SPLINE
SPL {X  -159.661, Y  +678.114, Z    +0.000, E1    -9.575, E3 +131003.511}
SPL {X  -159.942, Y  +672.020, Z    +0.000, E1    -4.692, E3 +131022.137}
SPL {X  -160.000, Y  +664.971, Z    +0.000, E1    +0.516, E3 +131041.688}
SPL {X  -160.000, Y  +660.032, Z    +0.000, E1    +3.995, E3 +131053.631}
SPL {X  -160.000, Y  +652.280, Z    +0.000, E1    +8.913, E3 +131072.146}
SPL {X  -160.000, Y  +644.147, Z    +0.000, E1   +13.158, E3 +131095.696}
SPL {X  -160.000, Y  +641.594, Z    +0.000, E1   +13.488, E3 +131114.137}
SPL {X  -160.000, Y  +639.799, Z    +0.000, E1   +13.486, E3 +131130.047}
SPL {X  -160.000, Y  +637.896, Z    +0.000, E1   +13.493, E3 +131146.862}
SPL {X  -160.000, Y  +635.832, Z    +0.000, E1   +13.499, E3 +131165.121}
SPL {X  -160.000, Y  +633.839, Z    +0.000, E1   +13.489, E3 +131182.810}
SPL {X  -160.000, Y  +631.625, Z    +0.000, E1   +13.508, E3 +131202.350}
SPL {X  -160.000, Y  +629.417, Z    +0.000, E1   +13.491, E3 +131221.962}
SPL {X  -160.000, Y  +627.180, Z    +0.000, E1   +13.508, E3 +131241.716}
SPL {X  -160.000, Y  +624.970, Z    +0.000, E1   +13.490, E3 +131261.366}
SPL {X  -160.000, Y  +623.020, Z    +0.000, E1   +13.491, E3 +131278.596}
SPL {X  -160.000, Y  +620.888, Z    +0.000, E1   +13.501, E3 +131297.458}
SPL {X  -160.000, Y  +618.790, Z    +0.000, E1   +13.488, E3 +131316.080}
SPL {X  -160.000, Y  +616.631, Z    +0.000, E1   +13.504, E3 +131335.134}
SPL {X  -160.000, Y  +614.230, Z    +0.000, E1   +13.510, E3 +131356.330}
SPL {X  -160.000, Y  +612.132, Z    +0.000, E1   +13.485, E3 +131375.046}
SPL {X  -160.000, Y  +610.405, Z    +0.000, E1   +13.477, E3 +131390.420}
SPL {X  -160.000, Y  +608.437, Z    +0.000, E1   +13.502, E3 +131407.675}
SPL {X  -160.000, Y  +606.281, Z    +0.000, E1   +13.502, E3 +131426.693}
SPL {X  -160.000, Y  +604.124, Z    +0.000, E1   +13.513, E3 +131445.748}
SPL {X  -160.000, Y  +601.878, Z    +0.000, E1   +13.505, E3 +131465.645}
SPL {X  -160.000, Y  +599.648, Z    +0.000, E1   +13.506, E3 +131485.422}
SPL {X  -160.000, Y  +597.673, Z    +0.000, E1   +13.479, E3 +131503.095}
SPL {X  -160.000, Y  +595.601, Z    +0.000, E1   +13.499, E3 +131521.379}
SPL {X  -160.000, Y  +593.187, Z    +0.000, E1   +13.500, E3 +131542.759}
SPL {X  -160.000, Y  +591.079, Z    +0.000, E1   +13.483, E3 +131561.485}
SPL {X  -160.000, Y  +589.151, Z    +0.000, E1   +13.489, E3 +131578.536}
SPL {X  -160.000, Y  +586.908, Z    +0.000, E1   +13.501, E3 +131598.381}
SPL {X  -160.000, Y  +584.660, Z    +0.000, E1   +13.490, E3 +131618.323}
SPL {X  -160.000, Y  +582.409, Z    +0.000, E1   +13.499, E3 +131638.241}
SPL {X  -160.000, Y  +580.150, Z    +0.000, E1   +13.490, E3 +131658.288}
SPL {X  -160.000, Y  +577.953, Z    +0.000, E1   +13.493, E3 +131677.746}
SPL {X  -160.000, Y  +575.630, Z    +0.000, E1   +13.502, E3 +131698.230}
SPL {X  -160.000, Y  +573.418, Z    +0.000, E1   +13.502, E3 +131717.738}
SPL {X  -160.000, Y  +571.226, Z    +0.000, E1   +13.520, E3 +131736.947}
SPL {X  -160.000, Y  +569.166, Z    +0.000, E1   +13.512, E3 +131755.137}
SPL {X  -160.000, Y  +567.275, Z    +0.000, E1   +13.517, E3 +131771.804}
SPL {X  -160.000, Y  +565.259, Z    +0.000, E1   +13.523, E3 +131789.593}
SPL {X  -160.000, Y  +563.305, Z    +0.000, E1   +13.512, E3 +131806.932}
SPL {X  -160.000, Y  +561.240, Z    +0.000, E1   +13.521, E3 +131825.193}
SPL {X  -160.000, Y  +558.881, Z    +0.000, E1   +13.524, E3 +131846.036}
SPL {X  -160.000, Y  +556.697, Z    +0.000, E1   +13.510, E3 +131865.422}
SPL {X  -160.000, Y  +554.624, Z    +0.000, E1   +13.512, E3 +131883.753}
SPL {X  -160.000, Y  +552.465, Z    +0.000, E1   +13.514, E3 +131902.837}
SPL {X  -160.000, Y  +550.315, Z    +0.000, E1   +13.514, E3 +131921.830}
SPL {X  -160.000, Y  +548.056, Z    +0.000, E1   +13.519, E3 +131941.831}
SPL {X  -160.000, Y  +545.826, Z    +0.000, E1   +13.501, E3 +131961.709}
SPL {X  -160.000, Y  +543.677, Z    +0.000, E1   +13.502, E3 +131980.767}
SPL {X  -160.000, Y  +541.664, Z    +0.000, E1   +13.489, E3 +131998.652}
SPL {X  -160.000, Y  +539.659, Z    +0.000, E1   +13.494, E3 +132016.413}
SPL {X  -160.000, Y  +537.370, Z    +0.000, E1   +13.501, E3 +132036.652}
SPL {X  -160.000, Y  +535.056, Z    +0.000, E1   +13.506, E3 +132057.047}
SPL {X  -160.000, Y  +532.975, Z    +0.000, E1   +13.494, E3 +132075.534}
SPL {X  -160.000, Y  +530.925, Z    +0.000, E1   +13.499, E3 +132093.696}
SPL {X  -160.000, Y  +528.768, Z    +0.000, E1   +13.498, E3 +132112.797}
SPL {X  -160.000, Y  +526.547, Z    +0.000, E1   +13.499, E3 +132132.466}
SPL {X  -160.000, Y  +523.964, Z    +0.000, E1   +13.742, E3 +132151.970}
SPL {X  -160.000, Y  +513.971, Z    +0.000, E1   +18.644, E3 +132170.882}
SPL {X  -160.000, Y  +513.562, Z    +0.000, E1   +16.972, E3 +132190.759}
SPL {X  -160.000, Y  +513.358, Z    +0.000, E1   +15.267, E3 +132211.031}
SPL {X  -160.000, Y  +512.244, Z    +0.000, E1   +14.473, E3 +132229.487}
SPL {X  -160.000, Y  +509.675, Z    +0.000, E1   +14.481, E3 +132250.631}
SPL {X  -160.000, Y  +507.162, Z    +0.000, E1   +14.470, E3 +132271.371}
SPL {X  -160.000, Y  +504.735, Z    +0.000, E1   +14.473, E3 +132291.342}
SPL {X  -160.000, Y  +502.261, Z    +0.000, E1   +14.476, E3 +132311.678}
SPL {X  -160.000, Y  +499.798, Z    +0.000, E1   +14.482, E3 +132331.880}
SPL {X  -160.000, Y  +497.435, Z    +0.000, E1   +14.476, E3 +132351.357}
SPL {X  -160.000, Y  +495.089, Z    +0.000, E1   +14.475, E3 +132370.724}
SPL {X  -160.000, Y  +492.764, Z    +0.000, E1   +14.469, E3 +132389.895}
SPL {X  -160.000, Y  +490.292, Z    +0.000, E1   +14.476, E3 +132410.296}
SPL {X  -160.000, Y  +487.641, Z    +0.000, E1   +14.470, E3 +132432.192}
SPL {X  -160.000, Y  +485.054, Z    +0.000, E1   +14.460, E3 +132453.635}
SPL {X  -160.000, Y  +482.421, Z    +0.000, E1   +14.461, E3 +132475.353}
SPL {X  -160.000, Y  +480.000, Z    +0.000, E1   +14.451, E3 +132495.318}
SPL {X  -160.000, Y  +477.551, Z    +0.000, E1   +14.466, E3 +132515.446}
SPL {X  -160.000, Y  +475.253, Z    +0.000, E1   +14.450, E3 +132534.420}
SPL {X  -160.000, Y  +473.070, Z    +0.000, E1   +14.454, E3 +132552.441}
SPL {X  -160.000, Y  +470.603, Z    +0.000, E1   +14.464, E3 +132572.741}
SPL {X  -160.000, Y  +468.243, Z    +0.000, E1   +14.458, E3 +132592.141}
SPL {X  -160.000, Y  +465.791, Z    +0.000, E1   +14.475, E3 +132612.285}
SPL {X  -160.000, Y  +463.103, Z    +0.000, E1   +14.474, E3 +132634.433}
SPL {X  -160.000, Y  +460.743, Z    +0.000, E1   +14.465, E3 +132653.842}
SPL {X  -160.000, Y  +458.292, Z    +0.000, E1   +14.492, E3 +132673.841}
SPL {X  -160.000, Y  +455.874, Z    +0.000, E1   +14.484, E3 +132693.699}
SPL {X  -160.000, Y  +453.555, Z    +0.000, E1   +14.488, E3 +132712.778}
SPL {X  -160.000, Y  +451.093, Z    +0.000, E1   +14.485, E3 +132733.090}
SPL {X  -160.000, Y  +448.700, Z    +0.000, E1   +14.483, E3 +132752.779}
SPL {X  -160.000, Y  +446.277, Z    +0.000, E1   +14.485, E3 +132772.703}
SPL {X  -160.000, Y  +443.879, Z    +0.000, E1   +14.485, E3 +132792.441}
SPL {X  -160.000, Y  +441.447, Z    +0.000, E1   +14.485, E3 +132812.448}
SPL {X  -160.000, Y  +439.006, Z    +0.000, E1   +14.488, E3 +132832.531}
SPL {X  -160.000, Y  +436.311, Z    +0.000, E1   +14.498, E3 +132854.690}
SPL {X  -160.000, Y  +433.559, Z    +0.000, E1   +14.491, E3 +132877.360}
SPL {X  -160.000, Y  +431.162, Z    +0.000, E1   +14.479, E3 +132897.111}
SPL {X  -160.000, Y  +429.152, Z    +0.000, E1   +14.469, E3 +132913.692}
SPL {X  -160.000, Y  +426.863, Z    +0.000, E1   +14.490, E3 +132932.471}
SPL {X  -160.000, Y  +424.653, Z    +0.000, E1   +14.467, E3 +132950.731}
SPL {X  -160.000, Y  +422.337, Z    +0.000, E1   +14.492, E3 +132969.715}
SPL {X  -160.000, Y  +419.639, Z    +0.000, E1   +14.504, E3 +132991.755}
SPL {X  -160.000, Y  +417.127, Z    +0.000, E1   +14.501, E3 +133012.346}
SPL {X  -160.000, Y  +414.849, Z    +0.000, E1   +14.496, E3 +133031.080}
SPL {X  -160.000, Y  +412.396, Z    +0.000, E1   +14.505, E3 +133051.269}
SPL {X  -160.000, Y  +409.815, Z    +0.000, E1   +14.498, E3 +133072.523}
SPL {X  -160.000, Y  +407.614, Z    +0.000, E1   +14.484, E3 +133090.649}
SPL {X  -160.000, Y  +405.406, Z    +0.000, E1   +14.501, E3 +133108.712}
SPL {X  -160.000, Y  +402.958, Z    +0.000, E1   +14.500, E3 +133128.882}
SPL {X  -160.000, Y  +400.690, Z    +0.000, E1   +14.484, E3 +133147.593}
SPL {X  -160.000, Y  +398.391, Z    +0.000, E1   +14.502, E3 +133166.419}
SPL {X  -160.000, Y  +395.999, Z    +0.000, E1   +14.484, E3 +133186.209}
SPL {X  -160.000, Y  +393.685, Z    +0.000, E1   +14.486, E3 +133205.282}
SPL {X  -159.999, Y  +391.313, Z    +0.000, E1   +14.479, E3 +133224.864}
SPL {X  -159.970, Y  +388.900, Z    +0.000, E1   +14.480, E3 +133244.748}
SPL {X  -159.903, Y  +386.417, Z    +0.000, E1   +14.475, E3 +133265.253}
SPL {X  -159.796, Y  +383.921, Z    +0.000, E1   +14.466, E3 +133285.909}
SPL {X  -159.651, Y  +381.443, Z    +0.000, E1   +14.453, E3 +133306.456}
SPL {X  -159.474, Y  +379.042, Z    +0.000, E1   +14.434, E3 +133326.420}
SPL {X  -159.316, Y  +377.219, Z    +0.000, E1   +14.400, E3 +133341.649}
ENDSPLINE

SPLINE
SPL {X  -159.452, Y  +378.767, Z    +0.000, E1   +11.887, E3 +133362.638}
SPL {X  -159.840, Y  +384.856, Z    +0.000, E1    +7.126, E3 +133381.609}
SPL {X  -159.991, Y  +390.336, Z    +0.000, E1    +2.803, E3 +133395.432}
SPL {X  -160.000, Y  +403.532, Z    +0.000, E1    -6.523, E3 +133413.153}
SPL {X  -160.000, Y  +409.023, Z    +0.000, E1   -10.003, E3 +133423.926}
SPL {X  -160.000, Y  +418.032, Z    +0.000, E1   -14.569, E3 +133448.786}
SPL {X  -160.000, Y  +420.561, Z    +0.000, E1   -14.816, E3 +133466.266}
SPL {X  -160.000, Y  +422.801, Z    +0.000, E1   -14.823, E3 +133484.214}
SPL {X  -160.000, Y  +425.518, Z    +0.000, E1   -14.845, E3 +133505.989}
SPL {X  -160.000, Y  +428.688, Z    +0.000, E1   -14.854, E3 +133531.397}
SPL {X  -160.000, Y  +431.971, Z    +0.000, E1   -14.849, E3 +133557.866}
SPL {X  -160.000, Y  +435.345, Z    +0.000, E1   -14.857, E3 +133584.916}
SPL {X  -160.000, Y  +438.732, Z    +0.000, E1   -14.858, E3 +133612.064}
SPL {X  -160.000, Y  +441.925, Z    +0.000, E1   -14.848, E3 +133637.734}
SPL {X  -160.000, Y  +444.299, Z    +0.000, E1   -14.809, E3 +133656.919}
SPL {X  -160.000, Y  +446.229, Z    +0.000, E1   -14.820, E3 +133672.338}
SPL {X  -160.000, Y  +448.987, Z    +0.000, E1   -14.868, E3 +133694.275}
SPL {X  -160.000, Y  +452.351, Z    +0.000, E1   -14.871, E3 +133721.251}
SPL {X  -160.000, Y  +455.709, Z    +0.000, E1   -14.880, E3 +133748.065}
SPL {X  -160.000, Y  +458.189, Z    +0.000, E1   -14.832, E3 +133768.067}
SPL {X  -160.000, Y  +459.885, Z    +0.000, E1   -14.825, E3 +133781.737}
SPL {X  -160.000, Y  +462.438, Z    +0.000, E1   -14.868, E3 +133802.147}
SPL {X  -160.000, Y  +465.575, Z    +0.000, E1   -14.849, E3 +133827.456}
SPL {X  -160.000, Y  +468.581, Z    +0.000, E1   -14.841, E3 +133851.688}
SPL {X  -160.000, Y  +471.795, Z    +0.000, E1   -14.854, E3 +133877.475}
SPL {X  -160.000, Y  +475.138, Z    +0.000, E1   -14.853, E3 +133904.326}
SPL {X  -160.000, Y  +477.981, Z    +0.000, E1   -14.823, E3 +133927.246}
SPL {X  -160.000, Y  +480.658, Z    +0.000, E1   -14.835, E3 +133948.722}
SPL {X  -160.000, Y  +483.534, Z    +0.000, E1   -14.838, E3 +133971.817}
SPL {X  -160.000, Y  +486.226, Z    +0.000, E1   -14.823, E3 +133993.482}
SPL {X  -160.000, Y  +488.751, Z    +0.000, E1   -14.827, E3 +134013.754}
SPL {X  -160.000, Y  +491.612, Z    +0.000, E1   -14.844, E3 +134036.677}
SPL {X  -160.000, Y  +494.417, Z    +0.000, E1   -14.827, E3 +134059.268}
SPL {X  -160.000, Y  +496.961, Z    +0.000, E1   -14.824, E3 +134079.712}
SPL {X  -160.000, Y  +499.610, Z    +0.000, E1   -14.830, E3 +134100.984}
SPL {X  -160.000, Y  +502.268, Z    +0.000, E1   -14.832, E3 +134122.254}
SPL {X  -160.000, Y  +505.041, Z    +0.000, E1   -14.849, E3 +134144.416}
SPL {X  -160.000, Y  +507.743, Z    +0.000, E1   -14.842, E3 +134166.040}
SPL {X  -160.000, Y  +510.437, Z    +0.000, E1   -14.860, E3 +134187.554}
SPL {X  -160.000, Y  +513.179, Z    +0.000, E1   -14.849, E3 +134209.601}
SPL {X  -160.000, Y  +515.613, Z    +0.000, E1   -14.829, E3 +134229.272}
SPL {X  -160.000, Y  +518.188, Z    +0.000, E1   -14.845, E3 +134249.901}
SPL {X  -160.000, Y  +520.790, Z    +0.000, E1   -14.839, E3 +134270.730}
SPL {X  -160.000, Y  +523.469, Z    +0.000, E1   -14.855, E3 +134292.178}
SPL {X  -160.000, Y  +526.403, Z    +0.000, E1   -14.858, E3 +134315.714}
SPL {X  -160.000, Y  +529.266, Z    +0.000, E1   -14.848, E3 +134338.722}
SPL {X  -160.000, Y  +531.688, Z    +0.000, E1   -14.826, E3 +134358.271}
SPL {X  -160.000, Y  +534.214, Z    +0.000, E1   -14.841, E3 +134378.534}
SPL {X  -160.000, Y  +537.002, Z    +0.000, E1   -14.839, E3 +134400.953}
SPL {X  -160.000, Y  +539.729, Z    +0.000, E1   -14.840, E3 +134422.764}
SPL {X  -160.000, Y  +542.408, Z    +0.000, E1   -14.839, E3 +134444.317}
SPL {X  -160.000, Y  +545.014, Z    +0.000, E1   -14.831, E3 +134465.262}
SPL {X  -160.000, Y  +547.659, Z    +0.000, E1   -14.839, E3 +134486.477}
SPL {X  -160.000, Y  +550.215, Z    +0.000, E1   -14.827, E3 +134507.042}
SPL {X  -160.000, Y  +552.762, Z    +0.000, E1   -14.836, E3 +134527.460}
SPL {X  -160.000, Y  +555.331, Z    +0.000, E1   -14.837, E3 +134548.001}
SPL {X  -160.000, Y  +558.235, Z    +0.000, E1   -14.869, E3 +134571.165}
SPL {X  -160.000, Y  +561.088, Z    +0.000, E1   -14.848, E3 +134594.083}
SPL {X  -160.000, Y  +563.693, Z    +0.000, E1   -14.852, E3 +134614.944}
SPL {X  -160.000, Y  +566.560, Z    +0.000, E1   -14.865, E3 +134637.921}
SPL {X  -160.000, Y  +569.305, Z    +0.000, E1   -14.848, E3 +134659.950}
SPL {X  -160.000, Y  +571.769, Z    +0.000, E1   -14.852, E3 +134679.696}
SPL {X  -160.000, Y  +574.366, Z    +0.000, E1   -14.855, E3 +134700.483}
SPL {X  -160.000, Y  +577.037, Z    +0.000, E1   -14.859, E3 +134721.882}
SPL {X  -160.000, Y  +579.855, Z    +0.000, E1   -14.869, E3 +134744.409}
SPL {X  -160.000, Y  +582.456, Z    +0.000, E1   -14.854, E3 +134765.269}
SPL {X  -160.000, Y  +585.083, Z    +0.000, E1   -14.866, E3 +134786.319}
SPL {X  -160.000, Y  +587.675, Z    +0.000, E1   -14.853, E3 +134807.110}
SPL {X  -160.000, Y  +590.216, Z    +0.000, E1   -14.864, E3 +134827.429}
SPL {X  -160.000, Y  +592.848, Z    +0.000, E1   -14.865, E3 +134848.480}
SPL {X  -160.000, Y  +595.342, Z    +0.000, E1   -14.848, E3 +134868.658}
SPL {X  -160.000, Y  +597.995, Z    +0.000, E1   -14.848, E3 +134889.998}
SPL {X  -160.000, Y  +600.731, Z    +0.000, E1   -14.846, E3 +134911.949}
SPL {X  -160.000, Y  +603.404, Z    +0.000, E1   -14.846, E3 +134933.385}
SPL {X  -160.000, Y  +605.923, Z    +0.000, E1   -14.838, E3 +134953.626}
SPL {X  -160.000, Y  +608.492, Z    +0.000, E1   -14.846, E3 +134974.230}
SPL {X  -160.000, Y  +611.345, Z    +0.000, E1   -14.856, E3 +134997.088}
SPL {X  -160.000, Y  +614.087, Z    +0.000, E1   -14.839, E3 +135019.147}
SPL {X  -160.000, Y  +616.566, Z    +0.000, E1   -14.839, E3 +135039.041}
SPL {X  -160.000, Y  +619.350, Z    +0.000, E1   -14.855, E3 +135061.329}
SPL {X  -160.000, Y  +622.198, Z    +0.000, E1   -14.846, E3 +135084.213}
SPL {X  -160.000, Y  +624.642, Z    +0.000, E1   -14.829, E3 +135103.886}
SPL {X  -160.000, Y  +627.119, Z    +0.000, E1   -14.843, E3 +135123.726}
SPL {X  -160.000, Y  +629.682, Z    +0.000, E1   -14.838, E3 +135144.295}
SPL {X  -160.000, Y  +632.223, Z    +0.000, E1   -14.841, E3 +135164.686}
SPL {X  -160.000, Y  +634.941, Z    +0.000, E1   -14.846, E3 +135186.484}
SPL {X  -160.000, Y  +637.723, Z    +0.000, E1   -14.844, E3 +135208.828}
SPL {X  -160.000, Y  +640.315, Z    +0.000, E1   -14.836, E3 +135229.626}
SPL {X  -160.000, Y  +643.085, Z    +0.000, E1   -14.865, E3 +135251.677}
SPL {X  -160.000, Y  +645.845, Z    +0.000, E1   -14.848, E3 +135273.865}
SPL {X  -160.000, Y  +648.229, Z    +0.000, E1   -14.834, E3 +135293.075}
SPL {X  -160.000, Y  +650.656, Z    +0.000, E1   -14.835, E3 +135312.631}
SPL {X  -160.000, Y  +653.134, Z    +0.000, E1   -14.827, E3 +135332.558}
SPL {X  -160.000, Y  +655.670, Z    +0.000, E1   -14.841, E3 +135352.852}
SPL {X  -160.000, Y  +658.349, Z    +0.000, E1   -14.842, E3 +135374.328}
SPL {X  -160.000, Y  +660.936, Z    +0.000, E1   -14.838, E3 +135395.080}
SPL {X  -160.000, Y  +663.567, Z    +0.000, E1   -14.845, E3 +135416.210}
SPL {X  -160.000, Y  +666.216, Z    +0.000, E1   -14.832, E3 +135437.527}
SPL {X  -159.997, Y  +668.731, Z    +0.000, E1   -14.834, E3 +135457.719}
SPL {X  -159.962, Y  +671.176, Z    +0.000, E1   -14.822, E3 +135477.430}
SPL {X  -159.895, Y  +673.507, Z    +0.000, E1   -14.821, E3 +135496.161}
SPL {X  -159.785, Y  +675.985, Z    +0.000, E1   -14.818, E3 +135516.163}
SPL {X  -159.627, Y  +678.622, Z    +0.000, E1   -14.804, E3 +135537.516}
SPL {X  -159.438, Y  +681.094, Z    +0.000, E1   -14.770, E3 +135557.687}
SPL {X  -159.262, Y  +683.054, Z    +0.000, E1   -14.719, E3 +135573.915}
ENDSPLINE

SPLINE
SPL {X  -159.661, Y  +678.114, Z    +0.000, E1    -9.575, E3 +135603.507}
SPL {X  -159.942, Y  +672.020, Z    +0.000, E1    -4.692, E3 +135622.134}
SPL {X  -160.000, Y  +664.971, Z    +0.000, E1    +0.516, E3 +135641.684}
SPL {X  -160.000, Y  +660.032, Z    +0.000, E1    +3.995, E3 +135653.627}
SPL {X  -160.000, Y  +652.280, Z    +0.000, E1    +8.913, E3 +135672.142}
SPL {X  -160.000, Y  +644.147, Z    +0.000, E1   +13.158, E3 +135695.693}
SPL {X  -160.000, Y  +641.594, Z    +0.000, E1   +13.488, E3 +135714.134}
SPL {X  -160.000, Y  +639.799, Z    +0.000, E1   +13.486, E3 +135730.044}
SPL {X  -160.000, Y  +637.896, Z    +0.000, E1   +13.493, E3 +135746.859}
SPL {X  -160.000, Y  +635.832, Z    +0.000, E1   +13.499, E3 +135765.118}
SPL {X  -160.000, Y  +633.839, Z    +0.000, E1   +13.489, E3 +135782.806}
SPL {X  -160.000, Y  +631.625, Z    +0.000, E1   +13.508, E3 +135802.347}
SPL {X  -160.000, Y  +629.417, Z    +0.000, E1   +13.491, E3 +135821.959}
SPL {X  -160.000, Y  +627.180, Z    +0.000, E1   +13.508, E3 +135841.713}
SPL {X  -160.000, Y  +624.970, Z    +0.000, E1   +13.490, E3 +135861.363}
SPL {X  -160.000, Y  +623.020, Z    +0.000, E1   +13.491, E3 +135878.592}
SPL {X  -160.000, Y  +620.888, Z    +0.000, E1   +13.501, E3 +135897.455}
SPL {X  -160.000, Y  +618.790, Z    +0.000, E1   +13.488, E3 +135916.077}
SPL {X  -160.000, Y  +616.631, Z    +0.000, E1   +13.504, E3 +135935.131}
SPL {X  -160.000, Y  +614.230, Z    +0.000, E1   +13.510, E3 +135956.327}
SPL {X  -160.000, Y  +612.132, Z    +0.000, E1   +13.485, E3 +135975.043}
SPL {X  -160.000, Y  +610.405, Z    +0.000, E1   +13.477, E3 +135990.416}
SPL {X  -160.000, Y  +608.437, Z    +0.000, E1   +13.502, E3 +136007.672}
SPL {X  -160.000, Y  +606.281, Z    +0.000, E1   +13.502, E3 +136026.689}
SPL {X  -160.000, Y  +604.124, Z    +0.000, E1   +13.513, E3 +136045.745}
SPL {X  -160.000, Y  +601.878, Z    +0.000, E1   +13.505, E3 +136065.642}
SPL {X  -160.000, Y  +599.648, Z    +0.000, E1   +13.506, E3 +136085.419}
SPL {X  -160.000, Y  +597.673, Z    +0.000, E1   +13.479, E3 +136103.092}
SPL {X  -160.000, Y  +595.601, Z    +0.000, E1   +13.499, E3 +136121.375}
SPL {X  -160.000, Y  +593.187, Z    +0.000, E1   +13.500, E3 +136142.755}
SPL {X  -160.000, Y  +591.079, Z    +0.000, E1   +13.483, E3 +136161.482}
SPL {X  -160.000, Y  +589.151, Z    +0.000, E1   +13.489, E3 +136178.533}
SPL {X  -160.000, Y  +586.908, Z    +0.000, E1   +13.501, E3 +136198.378}
SPL {X  -160.000, Y  +584.660, Z    +0.000, E1   +13.490, E3 +136218.320}
SPL {X  -160.000, Y  +582.409, Z    +0.000, E1   +13.499, E3 +136238.238}
SPL {X  -160.000, Y  +580.150, Z    +0.000, E1   +13.490, E3 +136258.284}
SPL {X  -160.000, Y  +577.953, Z    +0.000, E1   +13.493, E3 +136277.743}
SPL {X  -160.000, Y  +575.630, Z    +0.000, E1   +13.502, E3 +136298.227}
SPL {X  -160.000, Y  +573.418, Z    +0.000, E1   +13.502, E3 +136317.735}
SPL {X  -160.000, Y  +571.226, Z    +0.000, E1   +13.520, E3 +136336.943}
SPL {X  -160.000, Y  +569.166, Z    +0.000, E1   +13.512, E3 +136355.134}
SPL {X  -160.000, Y  +567.275, Z    +0.000, E1   +13.517, E3 +136371.801}
SPL {X  -160.000, Y  +565.259, Z    +0.000, E1   +13.523, E3 +136389.590}
SPL {X  -160.000, Y  +563.305, Z    +0.000, E1   +13.512, E3 +136406.929}
SPL {X  -160.000, Y  +561.240, Z    +0.000, E1   +13.521, E3 +136425.190}
SPL {X  -160.000, Y  +558.881, Z    +0.000, E1   +13.524, E3 +136446.032}
SPL {X  -160.000, Y  +556.697, Z    +0.000, E1   +13.510, E3 +136465.418}
SPL {X  -160.000, Y  +554.624, Z    +0.000, E1   +13.512, E3 +136483.749}
SPL {X  -160.000, Y  +552.465, Z    +0.000, E1   +13.514, E3 +136502.834}
SPL {X  -160.000, Y  +550.315, Z    +0.000, E1   +13.514, E3 +136521.827}
SPL {X  -160.000, Y  +548.056, Z    +0.000, E1   +13.519, E3 +136541.828}
SPL {X  -160.000, Y  +545.826, Z    +0.000, E1   +13.501, E3 +136561.706}
SPL {X  -160.000, Y  +543.677, Z    +0.000, E1   +13.502, E3 +136580.764}
SPL {X  -160.000, Y  +541.664, Z    +0.000, E1   +13.489, E3 +136598.649}
SPL {X  -160.000, Y  +539.659, Z    +0.000, E1   +13.494, E3 +136616.409}
SPL {X  -160.000, Y  +537.370, Z    +0.000, E1   +13.501, E3 +136636.648}
SPL {X  -160.000, Y  +535.056, Z    +0.000, E1   +13.506, E3 +136657.044}
SPL {X  -160.000, Y  +532.975, Z    +0.000, E1   +13.494, E3 +136675.531}
SPL {X  -160.000, Y  +530.925, Z    +0.000, E1   +13.499, E3 +136693.692}
SPL {X  -160.000, Y  +528.768, Z    +0.000, E1   +13.498, E3 +136712.794}
SPL {X  -160.000, Y  +526.547, Z    +0.000, E1   +13.499, E3 +136732.462}
SPL {X  -160.000, Y  +523.964, Z    +0.000, E1   +13.742, E3 +136751.967}
SPL {X  -160.000, Y  +513.971, Z    +0.000, E1   +18.644, E3 +136770.879}
SPL {X  -160.000, Y  +513.562, Z    +0.000, E1   +16.972, E3 +136790.756}
SPL {X  -160.000, Y  +513.358, Z    +0.000, E1   +15.267, E3 +136811.028}
SPL {X  -160.000, Y  +512.244, Z    +0.000, E1   +14.473, E3 +136829.484}
SPL {X  -160.000, Y  +509.675, Z    +0.000, E1   +14.481, E3 +136850.627}
SPL {X  -160.000, Y  +507.162, Z    +0.000, E1   +14.470, E3 +136871.367}
SPL {X  -160.000, Y  +504.735, Z    +0.000, E1   +14.473, E3 +136891.339}
SPL {X  -160.000, Y  +502.261, Z    +0.000, E1   +14.476, E3 +136911.675}
SPL {X  -160.000, Y  +499.798, Z    +0.000, E1   +14.482, E3 +136931.877}
SPL {X  -160.000, Y  +497.435, Z    +0.000, E1   +14.476, E3 +136951.354}
SPL {X  -160.000, Y  +495.089, Z    +0.000, E1   +14.475, E3 +136970.721}
SPL {X  -160.000, Y  +492.764, Z    +0.000, E1   +14.469, E3 +136989.892}
SPL {X  -160.000, Y  +490.292, Z    +0.000, E1   +14.476, E3 +137010.293}
SPL {X  -160.000, Y  +487.641, Z    +0.000, E1   +14.470, E3 +137032.189}
SPL {X  -160.000, Y  +485.054, Z    +0.000, E1   +14.460, E3 +137053.632}
SPL {X  -160.000, Y  +482.421, Z    +0.000, E1   +14.461, E3 +137075.350}
SPL {X  -160.000, Y  +480.000, Z    +0.000, E1   +14.451, E3 +137095.314}
SPL {X  -160.000, Y  +477.551, Z    +0.000, E1   +14.466, E3 +137115.443}
SPL {X  -160.000, Y  +475.253, Z    +0.000, E1   +14.450, E3 +137134.417}
SPL {X  -160.000, Y  +473.070, Z    +0.000, E1   +14.454, E3 +137152.438}
SPL {X  -160.000, Y  +470.603, Z    +0.000, E1   +14.464, E3 +137172.738}
SPL {X  -160.000, Y  +468.243, Z    +0.000, E1   +14.458, E3 +137192.137}
SPL {X  -160.000, Y  +465.791, Z    +0.000, E1   +14.475, E3 +137212.281}
SPL {X  -160.000, Y  +463.103, Z    +0.000, E1   +14.474, E3 +137234.430}
SPL {X  -160.000, Y  +460.743, Z    +0.000, E1   +14.465, E3 +137253.838}
SPL {X  -160.000, Y  +458.292, Z    +0.000, E1   +14.492, E3 +137273.838}
SPL {X  -160.000, Y  +455.874, Z    +0.000, E1   +14.484, E3 +137293.695}
SPL {X  -160.000, Y  +453.555, Z    +0.000, E1   +14.488, E3 +137312.775}
SPL {X  -160.000, Y  +451.093, Z    +0.000, E1   +14.485, E3 +137333.087}
SPL {X  -160.000, Y  +448.700, Z    +0.000, E1   +14.483, E3 +137352.776}
SPL {X  -160.000, Y  +446.277, Z    +0.000, E1   +14.485, E3 +137372.700}
SPL {X  -160.000, Y  +443.879, Z    +0.000, E1   +14.485, E3 +137392.438}
SPL {X  -160.000, Y  +441.447, Z    +0.000, E1   +14.485, E3 +137412.445}
SPL {X  -160.000, Y  +439.006, Z    +0.000, E1   +14.488, E3 +137432.528}
SPL {X  -160.000, Y  +436.311, Z    +0.000, E1   +14.498, E3 +137454.687}
SPL {X  -160.000, Y  +433.559, Z    +0.000, E1   +14.491, E3 +137477.357}
SPL {X  -160.000, Y  +431.162, Z    +0.000, E1   +14.479, E3 +137497.108}
SPL {X  -160.000, Y  +429.152, Z    +0.000, E1   +14.469, E3 +137513.689}
SPL {X  -160.000, Y  +426.863, Z    +0.000, E1   +14.490, E3 +137532.468}
SPL {X  -160.000, Y  +424.653, Z    +0.000, E1   +14.467, E3 +137550.728}
SPL {X  -160.000, Y  +422.337, Z    +0.000, E1   +14.492, E3 +137569.712}
SPL {X  -160.000, Y  +419.639, Z    +0.000, E1   +14.504, E3 +137591.752}
SPL {X  -160.000, Y  +417.127, Z    +0.000, E1   +14.501, E3 +137612.343}
SPL {X  -160.000, Y  +414.849, Z    +0.000, E1   +14.496, E3 +137631.077}
SPL {X  -160.000, Y  +412.396, Z    +0.000, E1   +14.505, E3 +137651.266}
SPL {X  -160.000, Y  +409.815, Z    +0.000, E1   +14.498, E3 +137672.520}
SPL {X  -160.000, Y  +407.614, Z    +0.000, E1   +14.484, E3 +137690.645}
SPL {X  -160.000, Y  +405.406, Z    +0.000, E1   +14.501, E3 +137708.708}
SPL {X  -160.000, Y  +402.958, Z    +0.000, E1   +14.500, E3 +137728.879}
SPL {X  -160.000, Y  +400.690, Z    +0.000, E1   +14.484, E3 +137747.590}
SPL {X  -160.000, Y  +398.391, Z    +0.000, E1   +14.502, E3 +137766.416}
SPL {X  -160.000, Y  +395.999, Z    +0.000, E1   +14.484, E3 +137786.206}
SPL {X  -160.000, Y  +393.685, Z    +0.000, E1   +14.486, E3 +137805.278}
SPL {X  -159.999, Y  +391.313, Z    +0.000, E1   +14.479, E3 +137824.860}
SPL {X  -159.970, Y  +388.900, Z    +0.000, E1   +14.480, E3 +137844.745}
SPL {X  -159.903, Y  +386.417, Z    +0.000, E1   +14.475, E3 +137865.250}
SPL {X  -159.796, Y  +383.921, Z    +0.000, E1   +14.466, E3 +137885.905}
SPL {X  -159.651, Y  +381.443, Z    +0.000, E1   +14.453, E3 +137906.453}
SPL {X  -159.474, Y  +379.042, Z    +0.000, E1   +14.434, E3 +137926.417}
SPL {X  -159.316, Y  +377.219, Z    +0.000, E1   +14.400, E3 +137941.645}
ENDSPLINE

SPLINE
SPL {X  -159.452, Y  +378.767, Z    +0.000, E1   +11.887, E3 +137962.635}
SPL {X  -159.840, Y  +384.856, Z    +0.000, E1    +7.126, E3 +137981.606}
SPL {X  -159.991, Y  +390.336, Z    +0.000, E1    +2.803, E3 +137995.429}
SPL {X  -160.000, Y  +403.532, Z    +0.000, E1    -6.523, E3 +138013.150}
SPL {X  -160.000, Y  +409.023, Z    +0.000, E1   -10.003, E3 +138023.923}
SPL {X  -160.000, Y  +418.032, Z    +0.000, E1   -14.569, E3 +138048.782}
SPL {X  -160.000, Y  +420.561, Z    +0.000, E1   -14.816, E3 +138066.263}
SPL {X  -160.000, Y  +422.801, Z    +0.000, E1   -14.823, E3 +138084.211}
SPL {X  -160.000, Y  +425.518, Z    +0.000, E1   -14.845, E3 +138105.986}
SPL {X  -160.000, Y  +428.688, Z    +0.000, E1   -14.854, E3 +138131.394}
SPL {X  -160.000, Y  +431.971, Z    +0.000, E1   -14.849, E3 +138157.862}
SPL {X  -160.000, Y  +435.345, Z    +0.000, E1   -14.857, E3 +138184.913}
SPL {X  -160.000, Y  +438.732, Z    +0.000, E1   -14.858, E3 +138212.061}
SPL {X  -160.000, Y  +441.925, Z    +0.000, E1   -14.848, E3 +138237.731}
SPL {X  -160.000, Y  +444.299, Z    +0.000, E1   -14.809, E3 +138256.916}
SPL {X  -160.000, Y  +446.229, Z    +0.000, E1   -14.820, E3 +138272.335}
SPL {X  -160.000, Y  +448.987, Z    +0.000, E1   -14.868, E3 +138294.272}
SPL {X  -160.000, Y  +452.351, Z    +0.000, E1   -14.871, E3 +138321.248}
SPL {X  -160.000, Y  +455.709, Z    +0.000, E1   -14.880, E3 +138348.062}
SPL {X  -160.000, Y  +458.189, Z    +0.000, E1   -14.832, E3 +138368.063}
SPL {X  -160.000, Y  +459.885, Z    +0.000, E1   -14.825, E3 +138381.734}
SPL {X  -160.000, Y  +462.438, Z    +0.000, E1   -14.868, E3 +138402.144}
SPL {X  -160.000, Y  +465.575, Z    +0.000, E1   -14.849, E3 +138427.452}
SPL {X  -160.000, Y  +468.581, Z    +0.000, E1   -14.841, E3 +138451.685}
SPL {X  -160.000, Y  +471.795, Z    +0.000, E1   -14.854, E3 +138477.472}
SPL {X  -160.000, Y  +475.138, Z    +0.000, E1   -14.853, E3 +138504.322}
SPL {X  -160.000, Y  +477.981, Z    +0.000, E1   -14.823, E3 +138527.243}
SPL {X  -160.000, Y  +480.658, Z    +0.000, E1   -14.835, E3 +138548.719}
SPL {X  -160.000, Y  +483.534, Z    +0.000, E1   -14.838, E3 +138571.814}
SPL {X  -160.000, Y  +486.226, Z    +0.000, E1   -14.823, E3 +138593.479}
SPL {X  -160.000, Y  +488.751, Z    +0.000, E1   -14.827, E3 +138613.751}
SPL {X  -160.000, Y  +491.612, Z    +0.000, E1   -14.844, E3 +138636.674}
SPL {X  -160.000, Y  +494.417, Z    +0.000, E1   -14.827, E3 +138659.265}
SPL {X  -160.000, Y  +496.961, Z    +0.000, E1   -14.824, E3 +138679.709}
SPL {X  -160.000, Y  +499.610, Z    +0.000, E1   -14.830, E3 +138700.981}
SPL {X  -160.000, Y  +502.268, Z    +0.000, E1   -14.832, E3 +138722.250}
SPL {X  -160.000, Y  +505.041, Z    +0.000, E1   -14.849, E3 +138744.413}
SPL {X  -160.000, Y  +507.743, Z    +0.000, E1   -14.842, E3 +138766.037}
SPL {X  -160.000, Y  +510.437, Z    +0.000, E1   -14.860, E3 +138787.551}
SPL {X  -160.000, Y  +513.179, Z    +0.000, E1   -14.849, E3 +138809.598}
SPL {X  -160.000, Y  +515.613, Z    +0.000, E1   -14.829, E3 +138829.268}
SPL {X  -160.000, Y  +518.188, Z    +0.000, E1   -14.845, E3 +138849.898}
SPL {X  -160.000, Y  +520.790, Z    +0.000, E1   -14.839, E3 +138870.727}
SPL {X  -160.000, Y  +523.469, Z    +0.000, E1   -14.855, E3 +138892.175}
SPL {X  -160.000, Y  +526.403, Z    +0.000, E1   -14.858, E3 +138915.711}
SPL {X  -160.000, Y  +529.266, Z    +0.000, E1   -14.848, E3 +138938.718}
SPL {X  -160.000, Y  +531.688, Z    +0.000, E1   -14.826, E3 +138958.268}
SPL {X  -160.000, Y  +534.214, Z    +0.000, E1   -14.841, E3 +138978.531}
SPL {X  -160.000, Y  +537.002, Z    +0.000, E1   -14.839, E3 +139000.949}
SPL {X  -160.000, Y  +539.729, Z    +0.000, E1   -14.840, E3 +139022.761}
SPL {X  -160.000, Y  +542.408, Z    +0.000, E1   -14.839, E3 +139044.314}
SPL {X  -160.000, Y  +545.014, Z    +0.000, E1   -14.831, E3 +139065.259}
SPL {X  -160.000, Y  +547.659, Z    +0.000, E1   -14.839, E3 +139086.474}
SPL {X  -160.000, Y  +550.215, Z    +0.000, E1   -14.827, E3 +139107.039}
SPL {X  -160.000, Y  +552.762, Z    +0.000, E1   -14.836, E3 +139127.457}
SPL {X  -160.000, Y  +555.331, Z    +0.000, E1   -14.837, E3 +139147.998}
SPL {X  -160.000, Y  +558.235, Z    +0.000, E1   -14.869, E3 +139171.161}
SPL {X  -160.000, Y  +561.088, Z    +0.000, E1   -14.848, E3 +139194.080}
SPL {X  -160.000, Y  +563.693, Z    +0.000, E1   -14.852, E3 +139214.940}
SPL {X  -160.000, Y  +566.560, Z    +0.000, E1   -14.865, E3 +139237.918}
SPL {X  -160.000, Y  +569.305, Z    +0.000, E1   -14.848, E3 +139259.947}
SPL {X  -160.000, Y  +571.769, Z    +0.000, E1   -14.852, E3 +139279.692}
SPL {X  -160.000, Y  +574.366, Z    +0.000, E1   -14.855, E3 +139300.479}
SPL {X  -160.000, Y  +577.037, Z    +0.000, E1   -14.859, E3 +139321.879}
SPL {X  -160.000, Y  +579.855, Z    +0.000, E1   -14.869, E3 +139344.406}
SPL {X  -160.000, Y  +582.456, Z    +0.000, E1   -14.854, E3 +139365.266}
SPL {X  -160.000, Y  +585.083, Z    +0.000, E1   -14.866, E3 +139386.316}
SPL {X  -160.000, Y  +587.675, Z    +0.000, E1   -14.853, E3 +139407.107}
SPL {X  -160.000, Y  +590.216, Z    +0.000, E1   -14.864, E3 +139427.426}
SPL {X  -160.000, Y  +592.848, Z    +0.000, E1   -14.865, E3 +139448.477}
SPL {X  -160.000, Y  +595.342, Z    +0.000, E1   -14.848, E3 +139468.655}
SPL {X  -160.000, Y  +597.995, Z    +0.000, E1   -14.848, E3 +139489.995}
SPL {X  -160.000, Y  +600.731, Z    +0.000, E1   -14.846, E3 +139511.946}
SPL {X  -160.000, Y  +603.404, Z    +0.000, E1   -14.846, E3 +139533.382}
SPL {X  -160.000, Y  +605.923, Z    +0.000, E1   -14.838, E3 +139553.623}
SPL {X  -160.000, Y  +608.492, Z    +0.000, E1   -14.846, E3 +139574.226}
SPL {X  -160.000, Y  +611.345, Z    +0.000, E1   -14.856, E3 +139597.085}
SPL {X  -160.000, Y  +614.087, Z    +0.000, E1   -14.839, E3 +139619.144}
SPL {X  -160.000, Y  +616.566, Z    +0.000, E1   -14.839, E3 +139639.038}
SPL {X  -160.000, Y  +619.350, Z    +0.000, E1   -14.855, E3 +139661.326}
SPL {X  -160.000, Y  +622.198, Z    +0.000, E1   -14.846, E3 +139684.210}
SPL {X  -160.000, Y  +624.642, Z    +0.000, E1   -14.829, E3 +139703.883}
SPL {X  -160.000, Y  +627.119, Z    +0.000, E1   -14.843, E3 +139723.723}
SPL {X  -160.000, Y  +629.682, Z    +0.000, E1   -14.838, E3 +139744.292}
SPL {X  -160.000, Y  +632.223, Z    +0.000, E1   -14.841, E3 +139764.683}
SPL {X  -160.000, Y  +634.941, Z    +0.000, E1   -14.846, E3 +139786.481}
SPL {X  -160.000, Y  +637.723, Z    +0.000, E1   -14.844, E3 +139808.825}
SPL {X  -160.000, Y  +640.315, Z    +0.000, E1   -14.836, E3 +139829.622}
SPL {X  -160.000, Y  +643.085, Z    +0.000, E1   -14.865, E3 +139851.674}
SPL {X  -160.000, Y  +645.845, Z    +0.000, E1   -14.848, E3 +139873.862}
SPL {X  -160.000, Y  +648.229, Z    +0.000, E1   -14.834, E3 +139893.072}
SPL {X  -160.000, Y  +650.656, Z    +0.000, E1   -14.835, E3 +139912.628}
SPL {X  -160.000, Y  +653.134, Z    +0.000, E1   -14.827, E3 +139932.555}
SPL {X  -160.000, Y  +655.670, Z    +0.000, E1   -14.841, E3 +139952.849}
SPL {X  -160.000, Y  +658.349, Z    +0.000, E1   -14.842, E3 +139974.325}
SPL {X  -160.000, Y  +660.936, Z    +0.000, E1   -14.838, E3 +139995.077}
SPL {X  -160.000, Y  +663.567, Z    +0.000, E1   -14.845, E3 +140016.207}
SPL {X  -160.000, Y  +666.216, Z    +0.000, E1   -14.832, E3 +140037.524}
SPL {X  -159.997, Y  +668.731, Z    +0.000, E1   -14.834, E3 +140057.716}
SPL {X  -159.962, Y  +671.176, Z    +0.000, E1   -14.822, E3 +140077.427}
SPL {X  -159.895, Y  +673.507, Z    +0.000, E1   -14.821, E3 +140096.158}
SPL {X  -159.785, Y  +675.985, Z    +0.000, E1   -14.818, E3 +140116.160}
SPL {X  -159.627, Y  +678.622, Z    +0.000, E1   -14.804, E3 +140137.512}
SPL {X  -159.438, Y  +681.094, Z    +0.000, E1   -14.770, E3 +140157.684}
SPL {X  -159.262, Y  +683.054, Z    +0.000, E1   -14.719, E3 +140173.912}
ENDSPLINE

SPLINE
SPL {X  -159.661, Y  +678.114, Z    +0.000, E1    -9.575, E3 +140203.504}
SPL {X  -159.942, Y  +672.020, Z    +0.000, E1    -4.692, E3 +140222.131}
SPL {X  -160.000, Y  +664.971, Z    +0.000, E1    +0.516, E3 +140241.681}
SPL {X  -160.000, Y  +660.032, Z    +0.000, E1    +3.995, E3 +140253.624}
SPL {X  -160.000, Y  +652.280, Z    +0.000, E1    +8.913, E3 +140272.139}
SPL {X  -160.000, Y  +644.147, Z    +0.000, E1   +13.158, E3 +140295.690}
SPL {X  -160.000, Y  +641.594, Z    +0.000, E1   +13.488, E3 +140314.131}
SPL {X  -160.000, Y  +639.799, Z    +0.000, E1   +13.486, E3 +140330.041}
SPL {X  -160.000, Y  +637.896, Z    +0.000, E1   +13.493, E3 +140346.856}
SPL {X  -160.000, Y  +635.832, Z    +0.000, E1   +13.499, E3 +140365.114}
SPL {X  -160.000, Y  +633.839, Z    +0.000, E1   +13.489, E3 +140382.803}
SPL {X  -160.000, Y  +631.625, Z    +0.000, E1   +13.508, E3 +140402.344}
SPL {X  -160.000, Y  +629.417, Z    +0.000, E1   +13.491, E3 +140421.955}
SPL {X  -160.000, Y  +627.180, Z    +0.000, E1   +13.508, E3 +140441.709}
SPL {X  -160.000, Y  +624.970, Z    +0.000, E1   +13.490, E3 +140461.359}
SPL {X  -160.000, Y  +623.020, Z    +0.000, E1   +13.491, E3 +140478.589}
SPL {X  -160.000, Y  +620.888, Z    +0.000, E1   +13.501, E3 +140497.452}
SPL {X  -160.000, Y  +618.790, Z    +0.000, E1   +13.488, E3 +140516.074}
SPL {X  -160.000, Y  +616.631, Z    +0.000, E1   +13.504, E3 +140535.128}
SPL {X  -160.000, Y  +614.230, Z    +0.000, E1   +13.510, E3 +140556.323}
SPL {X  -160.000, Y  +612.132, Z    +0.000, E1   +13.485, E3 +140575.040}
SPL {X  -160.000, Y  +610.405, Z    +0.000, E1   +13.477, E3 +140590.413}
SPL {X  -160.000, Y  +608.437, Z    +0.000, E1   +13.502, E3 +140607.669}
SPL {X  -160.000, Y  +606.281, Z    +0.000, E1   +13.502, E3 +140626.686}
SPL {X  -160.000, Y  +604.124, Z    +0.000, E1   +13.513, E3 +140645.741}
SPL {X  -160.000, Y  +601.878, Z    +0.000, E1   +13.505, E3 +140665.639}
SPL {X  -160.000, Y  +599.648, Z    +0.000, E1   +13.506, E3 +140685.415}
SPL {X  -160.000, Y  +597.673, Z    +0.000, E1   +13.479, E3 +140703.089}
SPL {X  -160.000, Y  +595.601, Z    +0.000, E1   +13.499, E3 +140721.372}
SPL {X  -160.000, Y  +593.187, Z    +0.000, E1   +13.500, E3 +140742.752}
SPL {X  -160.000, Y  +591.079, Z    +0.000, E1   +13.483, E3 +140761.478}
SPL {X  -160.000, Y  +589.151, Z    +0.000, E1   +13.489, E3 +140778.529}
SPL {X  -160.000, Y  +586.908, Z    +0.000, E1   +13.501, E3 +140798.375}
SPL {X  -160.000, Y  +584.660, Z    +0.000, E1   +13.490, E3 +140818.316}
SPL {X  -160.000, Y  +582.409, Z    +0.000, E1   +13.499, E3 +140838.235}
SPL {X  -160.000, Y  +580.150, Z    +0.000, E1   +13.490, E3 +140858.281}
SPL {X  -160.000, Y  +577.953, Z    +0.000, E1   +13.493, E3 +140877.739}
SPL {X  -160.000, Y  +575.630, Z    +0.000, E1   +13.502, E3 +140898.223}
SPL {X  -160.000, Y  +573.418, Z    +0.000, E1   +13.502, E3 +140917.731}
SPL {X  -160.000, Y  +571.226, Z    +0.000, E1   +13.520, E3 +140936.940}
SPL {X  -160.000, Y  +569.166, Z    +0.000, E1   +13.512, E3 +140955.131}
SPL {X  -160.000, Y  +567.275, Z    +0.000, E1   +13.517, E3 +140971.798}
SPL {X  -160.000, Y  +565.259, Z    +0.000, E1   +13.523, E3 +140989.587}
SPL {X  -160.000, Y  +563.305, Z    +0.000, E1   +13.512, E3 +141006.925}
SPL {X  -160.000, Y  +561.240, Z    +0.000, E1   +13.521, E3 +141025.187}
SPL {X  -160.000, Y  +558.881, Z    +0.000, E1   +13.524, E3 +141046.029}
SPL {X  -160.000, Y  +556.697, Z    +0.000, E1   +13.510, E3 +141065.415}
SPL {X  -160.000, Y  +554.624, Z    +0.000, E1   +13.512, E3 +141083.746}
SPL {X  -160.000, Y  +552.465, Z    +0.000, E1   +13.514, E3 +141102.830}
SPL {X  -160.000, Y  +550.315, Z    +0.000, E1   +13.514, E3 +141121.824}
SPL {X  -160.000, Y  +548.056, Z    +0.000, E1   +13.519, E3 +141141.825}
SPL {X  -160.000, Y  +545.826, Z    +0.000, E1   +13.501, E3 +141161.703}
SPL {X  -160.000, Y  +543.677, Z    +0.000, E1   +13.502, E3 +141180.761}
SPL {X  -160.000, Y  +541.664, Z    +0.000, E1   +13.489, E3 +141198.646}
SPL {X  -160.000, Y  +539.659, Z    +0.000, E1   +13.494, E3 +141216.406}
SPL {X  -160.000, Y  +537.370, Z    +0.000, E1   +13.501, E3 +141236.645}
SPL {X  -160.000, Y  +535.056, Z    +0.000, E1   +13.506, E3 +141257.041}
SPL {X  -160.000, Y  +532.975, Z    +0.000, E1   +13.494, E3 +141275.527}
SPL {X  -160.000, Y  +530.925, Z    +0.000, E1   +13.499, E3 +141293.689}
SPL {X  -160.000, Y  +528.768, Z    +0.000, E1   +13.498, E3 +141312.791}
SPL {X  -160.000, Y  +526.547, Z    +0.000, E1   +13.499, E3 +141332.459}
SPL {X  -160.000, Y  +523.964, Z    +0.000, E1   +13.742, E3 +141351.964}
SPL {X  -160.000, Y  +513.971, Z    +0.000, E1   +18.644, E3 +141370.876}
SPL {X  -160.000, Y  +513.562, Z    +0.000, E1   +16.972, E3 +141390.752}
SPL {X  -160.000, Y  +513.358, Z    +0.000, E1   +15.267, E3 +141411.024}
SPL {X  -160.000, Y  +512.244, Z    +0.000, E1   +14.473, E3 +141429.481}
SPL {X  -160.000, Y  +509.675, Z    +0.000, E1   +14.481, E3 +141450.624}
SPL {X  -160.000, Y  +507.162, Z    +0.000, E1   +14.470, E3 +141471.364}
SPL {X  -160.000, Y  +504.735, Z    +0.000, E1   +14.473, E3 +141491.336}
SPL {X  -160.000, Y  +502.261, Z    +0.000, E1   +14.476, E3 +141511.672}
SPL {X  -160.000, Y  +499.798, Z    +0.000, E1   +14.482, E3 +141531.874}
SPL {X  -160.000, Y  +497.435, Z    +0.000, E1   +14.476, E3 +141551.351}
SPL {X  -160.000, Y  +495.089, Z    +0.000, E1   +14.475, E3 +141570.717}
SPL {X  -160.000, Y  +492.764, Z    +0.000, E1   +14.469, E3 +141589.889}
SPL {X  -160.000, Y  +490.292, Z    +0.000, E1   +14.476, E3 +141610.290}
SPL {X  -160.000, Y  +487.641, Z    +0.000, E1   +14.470, E3 +141632.186}
SPL {X  -160.000, Y  +485.054, Z    +0.000, E1   +14.460, E3 +141653.629}
SPL {X  -160.000, Y  +482.421, Z    +0.000, E1   +14.461, E3 +141675.347}
SPL {X  -160.000, Y  +480.000, Z    +0.000, E1   +14.451, E3 +141695.311}
SPL {X  -160.000, Y  +477.551, Z    +0.000, E1   +14.466, E3 +141715.440}
SPL {X  -160.000, Y  +475.253, Z    +0.000, E1   +14.450, E3 +141734.414}
SPL {X  -160.000, Y  +473.070, Z    +0.000, E1   +14.454, E3 +141752.435}
SPL {X  -160.000, Y  +470.603, Z    +0.000, E1   +14.464, E3 +141772.735}
SPL {X  -160.000, Y  +468.243, Z    +0.000, E1   +14.458, E3 +141792.134}
SPL {X  -160.000, Y  +465.791, Z    +0.000, E1   +14.475, E3 +141812.278}
SPL {X  -160.000, Y  +463.103, Z    +0.000, E1   +14.474, E3 +141834.427}
SPL {X  -160.000, Y  +460.743, Z    +0.000, E1   +14.465, E3 +141853.835}
SPL {X  -160.000, Y  +458.292, Z    +0.000, E1   +14.492, E3 +141873.835}
SPL {X  -160.000, Y  +455.874, Z    +0.000, E1   +14.484, E3 +141893.692}
SPL {X  -160.000, Y  +453.555, Z    +0.000, E1   +14.488, E3 +141912.771}
SPL {X  -160.000, Y  +451.093, Z    +0.000, E1   +14.485, E3 +141933.084}
SPL {X  -160.000, Y  +448.700, Z    +0.000, E1   +14.483, E3 +141952.773}
SPL {X  -160.000, Y  +446.277, Z    +0.000, E1   +14.485, E3 +141972.697}
SPL {X  -160.000, Y  +443.879, Z    +0.000, E1   +14.485, E3 +141992.435}
SPL {X  -160.000, Y  +441.447, Z    +0.000, E1   +14.485, E3 +142012.442}
SPL {X  -160.000, Y  +439.006, Z    +0.000, E1   +14.488, E3 +142032.525}
SPL {X  -160.000, Y  +436.311, Z    +0.000, E1   +14.498, E3 +142054.684}
SPL {X  -160.000, Y  +433.559, Z    +0.000, E1   +14.491, E3 +142077.353}
SPL {X  -160.000, Y  +431.162, Z    +0.000, E1   +14.479, E3 +142097.105}
SPL {X  -160.000, Y  +429.152, Z    +0.000, E1   +14.469, E3 +142113.686}
SPL {X  -160.000, Y  +426.863, Z    +0.000, E1   +14.490, E3 +142132.465}
SPL {X  -160.000, Y  +424.653, Z    +0.000, E1   +14.467, E3 +142150.724}
SPL {X  -160.000, Y  +422.337, Z    +0.000, E1   +14.492, E3 +142169.709}
SPL {X  -160.000, Y  +419.639, Z    +0.000, E1   +14.504, E3 +142191.748}
SPL {X  -160.000, Y  +417.127, Z    +0.000, E1   +14.501, E3 +142212.340}
SPL {X  -160.000, Y  +414.849, Z    +0.000, E1   +14.496, E3 +142231.074}
SPL {X  -160.000, Y  +412.396, Z    +0.000, E1   +14.505, E3 +142251.263}
SPL {X  -160.000, Y  +409.815, Z    +0.000, E1   +14.498, E3 +142272.517}
SPL {X  -160.000, Y  +407.614, Z    +0.000, E1   +14.484, E3 +142290.642}
SPL {X  -160.000, Y  +405.406, Z    +0.000, E1   +14.501, E3 +142308.705}
SPL {X  -160.000, Y  +402.958, Z    +0.000, E1   +14.500, E3 +142328.875}
SPL {X  -160.000, Y  +400.690, Z    +0.000, E1   +14.484, E3 +142347.587}
SPL {X  -160.000, Y  +398.391, Z    +0.000, E1   +14.502, E3 +142366.413}
SPL {X  -160.000, Y  +395.999, Z    +0.000, E1   +14.484, E3 +142386.203}
SPL {X  -160.000, Y  +393.685, Z    +0.000, E1   +14.486, E3 +142405.275}
SPL {X  -159.999, Y  +391.313, Z    +0.000, E1   +14.479, E3 +142424.857}
SPL {X  -159.970, Y  +388.900, Z    +0.000, E1   +14.480, E3 +142444.741}
SPL {X  -159.903, Y  +386.417, Z    +0.000, E1   +14.475, E3 +142465.247}
SPL {X  -159.796, Y  +383.921, Z    +0.000, E1   +14.466, E3 +142485.902}
SPL {X  -159.651, Y  +381.443, Z    +0.000, E1   +14.453, E3 +142506.450}
SPL {X  -159.474, Y  +379.042, Z    +0.000, E1   +14.434, E3 +142526.414}
SPL {X  -159.316, Y  +377.219, Z    +0.000, E1   +14.400, E3 +142541.642}
ENDSPLINE

SPLINE
SPL {X  -159.452, Y  +378.767, Z    +0.000, E1   +11.887, E3 +142562.631}
SPL {X  -159.840, Y  +384.856, Z    +0.000, E1    +7.126, E3 +142581.603}
SPL {X  -159.991, Y  +390.336, Z    +0.000, E1    +2.803, E3 +142595.426}
SPL {X  -160.000, Y  +403.532, Z    +0.000, E1    -6.523, E3 +142613.146}
SPL {X  -160.000, Y  +409.023, Z    +0.000, E1   -10.003, E3 +142623.920}
SPL {X  -160.000, Y  +418.032, Z    +0.000, E1   -14.569, E3 +142648.779}
SPL {X  -160.000, Y  +420.561, Z    +0.000, E1   -14.816, E3 +142666.259}
SPL {X  -160.000, Y  +422.801, Z    +0.000, E1   -14.823, E3 +142684.208}
SPL {X  -160.000, Y  +425.518, Z    +0.000, E1   -14.845, E3 +142705.982}
SPL {X  -160.000, Y  +428.688, Z    +0.000, E1   -14.854, E3 +142731.391}
SPL {X  -160.000, Y  +431.971, Z    +0.000, E1   -14.849, E3 +142757.859}
SPL {X  -160.000, Y  +435.345, Z    +0.000, E1   -14.857, E3 +142784.909}
SPL {X  -160.000, Y  +438.732, Z    +0.000, E1   -14.858, E3 +142812.058}
SPL {X  -160.000, Y  +441.925, Z    +0.000, E1   -14.848, E3 +142837.728}
SPL {X  -160.000, Y  +444.299, Z    +0.000, E1   -14.809, E3 +142856.913}
SPL {X  -160.000, Y  +446.229, Z    +0.000, E1   -14.820, E3 +142872.332}
SPL {X  -160.000, Y  +448.987, Z    +0.000, E1   -14.868, E3 +142894.268}
SPL {X  -160.000, Y  +452.351, Z    +0.000, E1   -14.871, E3 +142921.244}
SPL {X  -160.000, Y  +455.709, Z    +0.000, E1   -14.880, E3 +142948.059}
SPL {X  -160.000, Y  +458.189, Z    +0.000, E1   -14.832, E3 +142968.060}
SPL {X  -160.000, Y  +459.885, Z    +0.000, E1   -14.825, E3 +142981.731}
SPL {X  -160.000, Y  +462.438, Z    +0.000, E1   -14.868, E3 +143002.141}
SPL {X  -160.000, Y  +465.575, Z    +0.000, E1   -14.849, E3 +143027.449}
SPL {X  -160.000, Y  +468.581, Z    +0.000, E1   -14.841, E3 +143051.681}
SPL {X  -160.000, Y  +471.795, Z    +0.000, E1   -14.854, E3 +143077.469}
SPL {X  -160.000, Y  +475.138, Z    +0.000, E1   -14.853, E3 +143104.319}
SPL {X  -160.000, Y  +477.981, Z    +0.000, E1   -14.823, E3 +143127.239}
SPL {X  -160.000, Y  +480.658, Z    +0.000, E1   -14.835, E3 +143148.716}
SPL {X  -160.000, Y  +483.534, Z    +0.000, E1   -14.838, E3 +143171.810}
SPL {X  -160.000, Y  +486.226, Z    +0.000, E1   -14.823, E3 +143193.475}
SPL {X  -160.000, Y  +488.751, Z    +0.000, E1   -14.827, E3 +143213.748}
SPL {X  -160.000, Y  +491.612, Z    +0.000, E1   -14.844, E3 +143236.671}
SPL {X  -160.000, Y  +494.417, Z    +0.000, E1   -14.827, E3 +143259.261}
SPL {X  -160.000, Y  +496.961, Z    +0.000, E1   -14.824, E3 +143279.705}
SPL {X  -160.000, Y  +499.610, Z    +0.000, E1   -14.830, E3 +143300.978}
SPL {X  -160.000, Y  +502.268, Z    +0.000, E1   -14.832, E3 +143322.247}
SPL {X  -160.000, Y  +505.041, Z    +0.000, E1   -14.849, E3 +143344.410}
SPL {X  -160.000, Y  +507.743, Z    +0.000, E1   -14.842, E3 +143366.034}
SPL {X  -160.000, Y  +510.437, Z    +0.000, E1   -14.860, E3 +143387.547}
SPL {X  -160.000, Y  +513.179, Z    +0.000, E1   -14.849, E3 +143409.595}
SPL {X  -160.000, Y  +515.613, Z    +0.000, E1   -14.829, E3 +143429.265}
SPL {X  -160.000, Y  +518.188, Z    +0.000, E1   -14.845, E3 +143449.895}
SPL {X  -160.000, Y  +520.790, Z    +0.000, E1   -14.839, E3 +143470.723}
SPL {X  -160.000, Y  +523.469, Z    +0.000, E1   -14.855, E3 +143492.172}
SPL {X  -160.000, Y  +526.403, Z    +0.000, E1   -14.858, E3 +143515.708}
SPL {X  -160.000, Y  +529.266, Z    +0.000, E1   -14.848, E3 +143538.715}
SPL {X  -160.000, Y  +531.688, Z    +0.000, E1   -14.826, E3 +143558.265}
SPL {X  -160.000, Y  +534.214, Z    +0.000, E1   -14.841, E3 +143578.528}
SPL {X  -160.000, Y  +537.002, Z    +0.000, E1   -14.839, E3 +143600.946}
SPL {X  -160.000, Y  +539.729, Z    +0.000, E1   -14.840, E3 +143622.758}
SPL {X  -160.000, Y  +542.408, Z    +0.000, E1   -14.839, E3 +143644.311}
SPL {X  -160.000, Y  +545.014, Z    +0.000, E1   -14.831, E3 +143665.256}
SPL {X  -160.000, Y  +547.659, Z    +0.000, E1   -14.839, E3 +143686.471}
SPL {X  -160.000, Y  +550.215, Z    +0.000, E1   -14.827, E3 +143707.036}
SPL {X  -160.000, Y  +552.762, Z    +0.000, E1   -14.836, E3 +143727.454}
SPL {X  -160.000, Y  +555.331, Z    +0.000, E1   -14.837, E3 +143747.995}
SPL {X  -160.000, Y  +558.235, Z    +0.000, E1   -14.869, E3 +143771.158}
SPL {X  -160.000, Y  +561.088, Z    +0.000, E1   -14.848, E3 +143794.077}
SPL {X  -160.000, Y  +563.693, Z    +0.000, E1   -14.852, E3 +143814.937}
SPL {X  -160.000, Y  +566.560, Z    +0.000, E1   -14.865, E3 +143837.915}
SPL {X  -160.000, Y  +569.305, Z    +0.000, E1   -14.848, E3 +143859.943}
SPL {X  -160.000, Y  +571.769, Z    +0.000, E1   -14.852, E3 +143879.689}
SPL {X  -160.000, Y  +574.366, Z    +0.000, E1   -14.855, E3 +143900.476}
SPL {X  -160.000, Y  +577.037, Z    +0.000, E1   -14.859, E3 +143921.876}
SPL {X  -160.000, Y  +579.855, Z    +0.000, E1   -14.869, E3 +143944.403}
SPL {X  -160.000, Y  +582.456, Z    +0.000, E1   -14.854, E3 +143965.263}
SPL {X  -160.000, Y  +585.083, Z    +0.000, E1   -14.866, E3 +143986.313}
SPL {X  -160.000, Y  +587.675, Z    +0.000, E1   -14.853, E3 +144007.104}
SPL {X  -160.000, Y  +590.216, Z    +0.000, E1   -14.864, E3 +144027.423}
SPL {X  -160.000, Y  +592.848, Z    +0.000, E1   -14.865, E3 +144048.474}
SPL {X  -160.000, Y  +595.342, Z    +0.000, E1   -14.848, E3 +144068.652}
SPL {X  -160.000, Y  +597.995, Z    +0.000, E1   -14.848, E3 +144089.991}
SPL {X  -160.000, Y  +600.731, Z    +0.000, E1   -14.846, E3 +144111.943}
SPL {X  -160.000, Y  +603.404, Z    +0.000, E1   -14.846, E3 +144133.379}
SPL {X  -160.000, Y  +605.923, Z    +0.000, E1   -14.838, E3 +144153.620}
SPL {X  -160.000, Y  +608.492, Z    +0.000, E1   -14.846, E3 +144174.223}
SPL {X  -160.000, Y  +611.345, Z    +0.000, E1   -14.856, E3 +144197.081}
SPL {X  -160.000, Y  +614.087, Z    +0.000, E1   -14.839, E3 +144219.141}
SPL {X  -160.000, Y  +616.566, Z    +0.000, E1   -14.839, E3 +144239.035}
SPL {X  -160.000, Y  +619.350, Z    +0.000, E1   -14.855, E3 +144261.323}
SPL {X  -160.000, Y  +622.198, Z    +0.000, E1   -14.846, E3 +144284.207}
SPL {X  -160.000, Y  +624.642, Z    +0.000, E1   -14.829, E3 +144303.880}
SPL {X  -160.000, Y  +627.119, Z    +0.000, E1   -14.843, E3 +144323.720}
SPL {X  -160.000, Y  +629.682, Z    +0.000, E1   -14.838, E3 +144344.289}
SPL {X  -160.000, Y  +632.223, Z    +0.000, E1   -14.841, E3 +144364.680}
SPL {X  -160.000, Y  +634.941, Z    +0.000, E1   -14.846, E3 +144386.477}
SPL {X  -160.000, Y  +637.723, Z    +0.000, E1   -14.844, E3 +144408.822}
SPL {X  -160.000, Y  +640.315, Z    +0.000, E1   -14.836, E3 +144429.619}
SPL {X  -160.000, Y  +643.085, Z    +0.000, E1   -14.865, E3 +144451.671}
SPL {X  -160.000, Y  +645.845, Z    +0.000, E1   -14.848, E3 +144473.859}
SPL {X  -160.000, Y  +648.229, Z    +0.000, E1   -14.834, E3 +144493.068}
SPL {X  -160.000, Y  +650.656, Z    +0.000, E1   -14.835, E3 +144512.625}
SPL {X  -160.000, Y  +653.134, Z    +0.000, E1   -14.827, E3 +144532.552}
SPL {X  -160.000, Y  +655.670, Z    +0.000, E1   -14.841, E3 +144552.846}
SPL {X  -160.000, Y  +658.349, Z    +0.000, E1   -14.842, E3 +144574.322}
SPL {X  -160.000, Y  +660.936, Z    +0.000, E1   -14.838, E3 +144595.074}
SPL {X  -160.000, Y  +663.567, Z    +0.000, E1   -14.845, E3 +144616.204}
SPL {X  -160.000, Y  +666.216, Z    +0.000, E1   -14.832, E3 +144637.520}
SPL {X  -159.997, Y  +668.731, Z    +0.000, E1   -14.834, E3 +144657.712}
SPL {X  -159.962, Y  +671.176, Z    +0.000, E1   -14.822, E3 +144677.424}
SPL {X  -159.895, Y  +673.507, Z    +0.000, E1   -14.821, E3 +144696.155}
SPL {X  -159.785, Y  +675.985, Z    +0.000, E1   -14.818, E3 +144716.156}
SPL {X  -159.627, Y  +678.622, Z    +0.000, E1   -14.804, E3 +144737.509}
SPL {X  -159.438, Y  +681.094, Z    +0.000, E1   -14.770, E3 +144757.681}
SPL {X  -159.262, Y  +683.054, Z    +0.000, E1   -14.719, E3 +144773.909}
ENDSPLINE

SPLINE
SPL {X  -159.661, Y  +678.114, Z    +0.000, E1    -9.575, E3 +144803.501}
SPL {X  -159.942, Y  +672.020, Z    +0.000, E1    -4.692, E3 +144822.128}
SPL {X  -160.000, Y  +664.971, Z    +0.000, E1    +0.516, E3 +144841.678}
SPL {X  -160.000, Y  +660.032, Z    +0.000, E1    +3.995, E3 +144853.621}
SPL {X  -160.000, Y  +652.280, Z    +0.000, E1    +8.913, E3 +144872.136}
SPL {X  -160.000, Y  +644.147, Z    +0.000, E1   +13.158, E3 +144895.686}
SPL {X  -160.000, Y  +641.594, Z    +0.000, E1   +13.488, E3 +144914.127}
SPL {X  -160.000, Y  +639.799, Z    +0.000, E1   +13.486, E3 +144930.037}
SPL {X  -160.000, Y  +637.896, Z    +0.000, E1   +13.493, E3 +144946.852}
SPL {X  -160.000, Y  +635.832, Z    +0.000, E1   +13.499, E3 +144965.111}
SPL {X  -160.000, Y  +633.839, Z    +0.000, E1   +13.489, E3 +144982.800}
SPL {X  -160.000, Y  +631.625, Z    +0.000, E1   +13.508, E3 +145002.341}
SPL {X  -160.000, Y  +629.417, Z    +0.000, E1   +13.491, E3 +145021.952}
SPL {X  -160.000, Y  +627.180, Z    +0.000, E1   +13.508, E3 +145041.706}
SPL {X  -160.000, Y  +624.970, Z    +0.000, E1   +13.490, E3 +145061.356}
SPL {X  -160.000, Y  +623.020, Z    +0.000, E1   +13.491, E3 +145078.586}
SPL {X  -160.000, Y  +620.888, Z    +0.000, E1   +13.501, E3 +145097.448}
SPL {X  -160.000, Y  +618.790, Z    +0.000, E1   +13.488, E3 +145116.071}
SPL {X  -160.000, Y  +616.631, Z    +0.000, E1   +13.504, E3 +145135.124}
SPL {X  -160.000, Y  +614.230, Z    +0.000, E1   +13.510, E3 +145156.320}
SPL {X  -160.000, Y  +612.132, Z    +0.000, E1   +13.485, E3 +145175.037}
SPL {X  -160.000, Y  +610.405, Z    +0.000, E1   +13.477, E3 +145190.410}
SPL {X  -160.000, Y  +608.437, Z    +0.000, E1   +13.502, E3 +145207.665}
SPL {X  -160.000, Y  +606.281, Z    +0.000, E1   +13.502, E3 +145226.683}
SPL {X  -160.000, Y  +604.124, Z    +0.000, E1   +13.513, E3 +145245.738}
SPL {X  -160.000, Y  +601.878, Z    +0.000, E1   +13.505, E3 +145265.635}
SPL {X  -160.000, Y  +599.648, Z    +0.000, E1   +13.506, E3 +145285.412}
SPL {X  -160.000, Y  +597.673, Z    +0.000, E1   +13.479, E3 +145303.086}
SPL {X  -160.000, Y  +595.601, Z    +0.000, E1   +13.499, E3 +145321.369}
SPL {X  -160.000, Y  +593.187, Z    +0.000, E1   +13.500, E3 +145342.749}
SPL {X  -160.000, Y  +591.079, Z    +0.000, E1   +13.483, E3 +145361.475}
SPL {X  -160.000, Y  +589.151, Z    +0.000, E1   +13.489, E3 +145378.526}
SPL {X  -160.000, Y  +586.908, Z    +0.000, E1   +13.501, E3 +145398.372}
SPL {X  -160.000, Y  +584.660, Z    +0.000, E1   +13.490, E3 +145418.313}
SPL {X  -160.000, Y  +582.409, Z    +0.000, E1   +13.499, E3 +145438.231}
SPL {X  -160.000, Y  +580.150, Z    +0.000, E1   +13.490, E3 +145458.278}
SPL {X  -160.000, Y  +577.953, Z    +0.000, E1   +13.493, E3 +145477.736}
SPL {X  -160.000, Y  +575.630, Z    +0.000, E1   +13.502, E3 +145498.220}
SPL {X  -160.000, Y  +573.418, Z    +0.000, E1   +13.502, E3 +145517.728}
SPL {X  -160.000, Y  +571.226, Z    +0.000, E1   +13.520, E3 +145536.937}
SPL {X  -160.000, Y  +569.166, Z    +0.000, E1   +13.512, E3 +145555.127}
SPL {X  -160.000, Y  +567.275, Z    +0.000, E1   +13.517, E3 +145571.795}
SPL {X  -160.000, Y  +565.259, Z    +0.000, E1   +13.523, E3 +145589.584}
SPL {X  -160.000, Y  +563.305, Z    +0.000, E1   +13.512, E3 +145606.922}
SPL {X  -160.000, Y  +561.240, Z    +0.000, E1   +13.521, E3 +145625.184}
SPL {X  -160.000, Y  +558.881, Z    +0.000, E1   +13.524, E3 +145646.026}
SPL {X  -160.000, Y  +556.697, Z    +0.000, E1   +13.510, E3 +145665.412}
SPL {X  -160.000, Y  +554.624, Z    +0.000, E1   +13.512, E3 +145683.743}
SPL {X  -160.000, Y  +552.465, Z    +0.000, E1   +13.514, E3 +145702.827}
SPL {X  -160.000, Y  +550.315, Z    +0.000, E1   +13.514, E3 +145721.821}
SPL {X  -160.000, Y  +548.056, Z    +0.000, E1   +13.519, E3 +145741.822}
SPL {X  -160.000, Y  +545.826, Z    +0.000, E1   +13.501, E3 +145761.700}
SPL {X  -160.000, Y  +543.677, Z    +0.000, E1   +13.502, E3 +145780.757}
SPL {X  -160.000, Y  +541.664, Z    +0.000, E1   +13.489, E3 +145798.643}
SPL {X  -160.000, Y  +539.659, Z    +0.000, E1   +13.494, E3 +145816.403}
SPL {X  -160.000, Y  +537.370, Z    +0.000, E1   +13.501, E3 +145836.642}
SPL {X  -160.000, Y  +535.056, Z    +0.000, E1   +13.506, E3 +145857.038}
SPL {X  -160.000, Y  +532.975, Z    +0.000, E1   +13.494, E3 +145875.524}
SPL {X  -160.000, Y  +530.925, Z    +0.000, E1   +13.499, E3 +145893.686}
SPL {X  -160.000, Y  +528.768, Z    +0.000, E1   +13.498, E3 +145912.787}
SPL {X  -160.000, Y  +526.547, Z    +0.000, E1   +13.499, E3 +145932.456}
SPL {X  -160.000, Y  +523.964, Z    +0.000, E1   +13.742, E3 +145951.961}
SPL {X  -160.000, Y  +513.971, Z    +0.000, E1   +18.644, E3 +145970.873}
SPL {X  -160.000, Y  +513.562, Z    +0.000, E1   +16.972, E3 +145990.749}
SPL {X  -160.000, Y  +513.358, Z    +0.000, E1   +15.267, E3 +146011.021}
SPL {X  -160.000, Y  +512.244, Z    +0.000, E1   +14.473, E3 +146029.478}
SPL {X  -160.000, Y  +509.675, Z    +0.000, E1   +14.481, E3 +146050.621}
SPL {X  -160.000, Y  +507.162, Z    +0.000, E1   +14.470, E3 +146071.361}
SPL {X  -160.000, Y  +504.735, Z    +0.000, E1   +14.473, E3 +146091.332}
SPL {X  -160.000, Y  +502.261, Z    +0.000, E1   +14.476, E3 +146111.668}
SPL {X  -160.000, Y  +499.798, Z    +0.000, E1   +14.482, E3 +146131.871}
SPL {X  -160.000, Y  +497.435, Z    +0.000, E1   +14.476, E3 +146151.347}
SPL {X  -160.000, Y  +495.089, Z    +0.000, E1   +14.475, E3 +146170.714}
SPL {X  -160.000, Y  +492.764, Z    +0.000, E1   +14.469, E3 +146189.886}
SPL {X  -160.000, Y  +490.292, Z    +0.000, E1   +14.476, E3 +146210.287}
SPL {X  -160.000, Y  +487.641, Z    +0.000, E1   +14.470, E3 +146232.183}
SPL {X  -160.000, Y  +485.054, Z    +0.000, E1   +14.460, E3 +146253.625}
SPL {X  -160.000, Y  +482.421, Z    +0.000, E1   +14.461, E3 +146275.344}
SPL {X  -160.000, Y  +480.000, Z    +0.000, E1   +14.451, E3 +146295.308}
SPL {X  -160.000, Y  +477.551, Z    +0.000, E1   +14.466, E3 +146315.436}
SPL {X  -160.000, Y  +475.253, Z    +0.000, E1   +14.450, E3 +146334.411}
SPL {X  -160.000, Y  +473.070, Z    +0.000, E1   +14.454, E3 +146352.432}
SPL {X  -160.000, Y  +470.603, Z    +0.000, E1   +14.464, E3 +146372.732}
SPL {X  -160.000, Y  +468.243, Z    +0.000, E1   +14.458, E3 +146392.131}
SPL {X  -160.000, Y  +465.791, Z    +0.000, E1   +14.475, E3 +146412.275}
SPL {X  -160.000, Y  +463.103, Z    +0.000, E1   +14.474, E3 +146434.424}
SPL {X  -160.000, Y  +460.743, Z    +0.000, E1   +14.465, E3 +146453.832}
SPL {X  -160.000, Y  +458.292, Z    +0.000, E1   +14.492, E3 +146473.831}
SPL {X  -160.000, Y  +455.874, Z    +0.000, E1   +14.484, E3 +146493.689}
SPL {X  -160.000, Y  +453.555, Z    +0.000, E1   +14.488, E3 +146512.768}
SPL {X  -160.000, Y  +451.093, Z    +0.000, E1   +14.485, E3 +146533.080}
SPL {X  -160.000, Y  +448.700, Z    +0.000, E1   +14.483, E3 +146552.770}
SPL {X  -160.000, Y  +446.277, Z    +0.000, E1   +14.485, E3 +146572.693}
SPL {X  -160.000, Y  +443.879, Z    +0.000, E1   +14.485, E3 +146592.432}
SPL {X  -160.000, Y  +441.447, Z    +0.000, E1   +14.485, E3 +146612.439}
SPL {X  -160.000, Y  +439.006, Z    +0.000, E1   +14.488, E3 +146632.522}
SPL {X  -160.000, Y  +436.311, Z    +0.000, E1   +14.498, E3 +146654.681}
SPL {X  -160.000, Y  +433.559, Z    +0.000, E1   +14.491, E3 +146677.350}
SPL {X  -160.000, Y  +431.162, Z    +0.000, E1   +14.479, E3 +146697.101}
SPL {X  -160.000, Y  +429.152, Z    +0.000, E1   +14.469, E3 +146713.683}
SPL {X  -160.000, Y  +426.863, Z    +0.000, E1   +14.490, E3 +146732.462}
SPL {X  -160.000, Y  +424.653, Z    +0.000, E1   +14.467, E3 +146750.721}
SPL {X  -160.000, Y  +422.337, Z    +0.000, E1   +14.492, E3 +146769.705}
SPL {X  -160.000, Y  +419.639, Z    +0.000, E1   +14.504, E3 +146791.745}
SPL {X  -160.000, Y  +417.127, Z    +0.000, E1   +14.501, E3 +146812.337}
SPL {X  -160.000, Y  +414.849, Z    +0.000, E1   +14.496, E3 +146831.071}
SPL {X  -160.000, Y  +412.396, Z    +0.000, E1   +14.505, E3 +146851.260}
SPL {X  -160.000, Y  +409.815, Z    +0.000, E1   +14.498, E3 +146872.514}
SPL {X  -160.000, Y  +407.614, Z    +0.000, E1   +14.484, E3 +146890.639}
SPL {X  -160.000, Y  +405.406, Z    +0.000, E1   +14.501, E3 +146908.702}
SPL {X  -160.000, Y  +402.958, Z    +0.000, E1   +14.500, E3 +146928.872}
SPL {X  -160.000, Y  +400.690, Z    +0.000, E1   +14.484, E3 +146947.584}
SPL {X  -160.000, Y  +398.391, Z    +0.000, E1   +14.502, E3 +146966.410}
SPL {X  -160.000, Y  +395.999, Z    +0.000, E1   +14.484, E3 +146986.200}
SPL {X  -160.000, Y  +393.685, Z    +0.000, E1   +14.486, E3 +147005.272}
SPL {X  -159.999, Y  +391.313, Z    +0.000, E1   +14.479, E3 +147024.854}
SPL {X  -159.970, Y  +388.900, Z    +0.000, E1   +14.480, E3 +147044.738}
SPL {X  -159.903, Y  +386.417, Z    +0.000, E1   +14.475, E3 +147065.243}
SPL {X  -159.796, Y  +383.921, Z    +0.000, E1   +14.466, E3 +147085.899}
SPL {X  -159.651, Y  +381.443, Z    +0.000, E1   +14.453, E3 +147106.446}
SPL {X  -159.474, Y  +379.042, Z    +0.000, E1   +14.434, E3 +147126.411}
SPL {X  -159.316, Y  +377.219, Z    +0.000, E1   +14.400, E3 +147141.639}
ENDSPLINE

SPLINE
SPL {X  -159.452, Y  +378.767, Z    +0.000, E1   +11.887, E3 +147162.628}
SPL {X  -159.840, Y  +384.856, Z    +0.000, E1    +7.126, E3 +147181.600}
SPL {X  -159.991, Y  +390.336, Z    +0.000, E1    +2.803, E3 +147195.423}
SPL {X  -160.000, Y  +403.532, Z    +0.000, E1    -6.523, E3 +147213.143}
SPL {X  -160.000, Y  +409.023, Z    +0.000, E1   -10.003, E3 +147223.917}
SPL {X  -160.000, Y  +418.032, Z    +0.000, E1   -14.569, E3 +147248.776}
SPL {X  -160.000, Y  +420.561, Z    +0.000, E1   -14.816, E3 +147266.256}
SPL {X  -160.000, Y  +422.801, Z    +0.000, E1   -14.823, E3 +147284.205}
SPL {X  -160.000, Y  +425.518, Z    +0.000, E1   -14.845, E3 +147305.979}
SPL {X  -160.000, Y  +428.688, Z    +0.000, E1   -14.854, E3 +147331.387}
SPL {X  -160.000, Y  +431.971, Z    +0.000, E1   -14.849, E3 +147357.856}
SPL {X  -160.000, Y  +435.345, Z    +0.000, E1   -14.857, E3 +147384.906}
SPL {X  -160.000, Y  +438.732, Z    +0.000, E1   -14.858, E3 +147412.055}
SPL {X  -160.000, Y  +441.925, Z    +0.000, E1   -14.848, E3 +147437.725}
SPL {X  -160.000, Y  +444.299, Z    +0.000, E1   -14.809, E3 +147456.910}
SPL {X  -160.000, Y  +446.229, Z    +0.000, E1   -14.820, E3 +147472.329}
SPL {X  -160.000, Y  +448.987, Z    +0.000, E1   -14.868, E3 +147494.265}
SPL {X  -160.000, Y  +452.351, Z    +0.000, E1   -14.871, E3 +147521.241}
SPL {X  -160.000, Y  +455.709, Z    +0.000, E1   -14.880, E3 +147548.055}
SPL {X  -160.000, Y  +458.189, Z    +0.000, E1   -14.832, E3 +147568.057}
SPL {X  -160.000, Y  +459.885, Z    +0.000, E1   -14.825, E3 +147581.728}
SPL {X  -160.000, Y  +462.438, Z    +0.000, E1   -14.868, E3 +147602.138}
SPL {X  -160.000, Y  +465.575, Z    +0.000, E1   -14.849, E3 +147627.446}
SPL {X  -160.000, Y  +468.581, Z    +0.000, E1   -14.841, E3 +147651.678}
SPL {X  -160.000, Y  +471.795, Z    +0.000, E1   -14.854, E3 +147677.466}
SPL {X  -160.000, Y  +475.138, Z    +0.000, E1   -14.853, E3 +147704.316}
SPL {X  -160.000, Y  +477.981, Z    +0.000, E1   -14.823, E3 +147727.236}
SPL {X  -160.000, Y  +480.658, Z    +0.000, E1   -14.835, E3 +147748.712}
SPL {X  -160.000, Y  +483.534, Z    +0.000, E1   -14.838, E3 +147771.807}
SPL {X  -160.000, Y  +486.226, Z    +0.000, E1   -14.823, E3 +147793.472}
SPL {X  -160.000, Y  +488.751, Z    +0.000, E1   -14.827, E3 +147813.745}
SPL {X  -160.000, Y  +491.612, Z    +0.000, E1   -14.844, E3 +147836.667}
SPL {X  -160.000, Y  +494.417, Z    +0.000, E1   -14.827, E3 +147859.258}
SPL {X  -160.000, Y  +496.961, Z    +0.000, E1   -14.824, E3 +147879.702}
SPL {X  -160.000, Y  +499.610, Z    +0.000, E1   -14.830, E3 +147900.975}
SPL {X  -160.000, Y  +502.268, Z    +0.000, E1   -14.832, E3 +147922.244}
SPL {X  -160.000, Y  +505.041, Z    +0.000, E1   -14.849, E3 +147944.407}
SPL {X  -160.000, Y  +507.743, Z    +0.000, E1   -14.842, E3 +147966.030}
SPL {X  -160.000, Y  +510.437, Z    +0.000, E1   -14.860, E3 +147987.544}
SPL {X  -160.000, Y  +513.179, Z    +0.000, E1   -14.849, E3 +148009.592}
SPL {X  -160.000, Y  +515.613, Z    +0.000, E1   -14.829, E3 +148029.262}
SPL {X  -160.000, Y  +518.188, Z    +0.000, E1   -14.845, E3 +148049.891}
SPL {X  -160.000, Y  +520.790, Z    +0.000, E1   -14.839, E3 +148070.720}
SPL {X  -160.000, Y  +523.469, Z    +0.000, E1   -14.855, E3 +148092.168}
SPL {X  -160.000, Y  +526.403, Z    +0.000, E1   -14.858, E3 +148115.705}
SPL {X  -160.000, Y  +529.266, Z    +0.000, E1   -14.848, E3 +148138.712}
SPL {X  -160.000, Y  +531.688, Z    +0.000, E1   -14.826, E3 +148158.262}
SPL {X  -160.000, Y  +534.214, Z    +0.000, E1   -14.841, E3 +148178.525}
SPL {X  -160.000, Y  +537.002, Z    +0.000, E1   -14.839, E3 +148200.943}
SPL {X  -160.000, Y  +539.729, Z    +0.000, E1   -14.840, E3 +148222.755}
SPL {X  -160.000, Y  +542.408, Z    +0.000, E1   -14.839, E3 +148244.308}
SPL {X  -160.000, Y  +545.014, Z    +0.000, E1   -14.831, E3 +148265.253}
SPL {X  -160.000, Y  +547.659, Z    +0.000, E1   -14.839, E3 +148286.467}
SPL {X  -160.000, Y  +550.215, Z    +0.000, E1   -14.827, E3 +148307.032}
SPL {X  -160.000, Y  +552.762, Z    +0.000, E1   -14.836, E3 +148327.451}
SPL {X  -160.000, Y  +555.331, Z    +0.000, E1   -14.837, E3 +148347.992}
SPL {X  -160.000, Y  +558.235, Z    +0.000, E1   -14.869, E3 +148371.155}
SPL {X  -160.000, Y  +561.088, Z    +0.000, E1   -14.848, E3 +148394.074}
SPL {X  -160.000, Y  +563.693, Z    +0.000, E1   -14.852, E3 +148414.934}
SPL {X  -160.000, Y  +566.560, Z    +0.000, E1   -14.865, E3 +148437.912}
SPL {X  -160.000, Y  +569.305, Z    +0.000, E1   -14.848, E3 +148459.940}
SPL {X  -160.000, Y  +571.769, Z    +0.000, E1   -14.852, E3 +148479.686}
SPL {X  -160.000, Y  +574.366, Z    +0.000, E1   -14.855, E3 +148500.473}
SPL {X  -160.000, Y  +577.037, Z    +0.000, E1   -14.859, E3 +148521.873}
SPL {X  -160.000, Y  +579.855, Z    +0.000, E1   -14.869, E3 +148544.400}
SPL {X  -160.000, Y  +582.456, Z    +0.000, E1   -14.854, E3 +148565.260}
SPL {X  -160.000, Y  +585.083, Z    +0.000, E1   -14.866, E3 +148586.309}
SPL {X  -160.000, Y  +587.675, Z    +0.000, E1   -14.853, E3 +148607.100}
SPL {X  -160.000, Y  +590.216, Z    +0.000, E1   -14.864, E3 +148627.420}
SPL {X  -160.000, Y  +592.848, Z    +0.000, E1   -14.865, E3 +148648.471}
SPL {X  -160.000, Y  +595.342, Z    +0.000, E1   -14.848, E3 +148668.648}
SPL {X  -160.000, Y  +597.995, Z    +0.000, E1   -14.848, E3 +148689.988}
SPL {X  -160.000, Y  +600.731, Z    +0.000, E1   -14.846, E3 +148711.940}
SPL {X  -160.000, Y  +603.404, Z    +0.000, E1   -14.846, E3 +148733.376}
SPL {X  -160.000, Y  +605.923, Z    +0.000, E1   -14.838, E3 +148753.616}
SPL {X  -160.000, Y  +608.492, Z    +0.000, E1   -14.846, E3 +148774.220}
SPL {X  -160.000, Y  +611.345, Z    +0.000, E1   -14.856, E3 +148797.078}
SPL {X  -160.000, Y  +614.087, Z    +0.000, E1   -14.839, E3 +148819.138}
SPL {X  -160.000, Y  +616.566, Z    +0.000, E1   -14.839, E3 +148839.031}
SPL {X  -160.000, Y  +619.350, Z    +0.000, E1   -14.855, E3 +148861.319}
SPL {X  -160.000, Y  +622.198, Z    +0.000, E1   -14.846, E3 +148884.204}
SPL {X  -160.000, Y  +624.642, Z    +0.000, E1   -14.829, E3 +148903.877}
SPL {X  -160.000, Y  +627.119, Z    +0.000, E1   -14.843, E3 +148923.716}
SPL {X  -160.000, Y  +629.682, Z    +0.000, E1   -14.838, E3 +148944.285}
SPL {X  -160.000, Y  +632.223, Z    +0.000, E1   -14.841, E3 +148964.677}
SPL {X  -160.000, Y  +634.941, Z    +0.000, E1   -14.846, E3 +148986.474}
SPL {X  -160.000, Y  +637.723, Z    +0.000, E1   -14.844, E3 +149008.818}
SPL {X  -160.000, Y  +640.315, Z    +0.000, E1   -14.836, E3 +149029.616}
SPL {X  -160.000, Y  +643.085, Z    +0.000, E1   -14.865, E3 +149051.668}
SPL {X  -160.000, Y  +645.845, Z    +0.000, E1   -14.848, E3 +149073.856}
SPL {X  -160.000, Y  +648.229, Z    +0.000, E1   -14.834, E3 +149093.065}
SPL {X  -160.000, Y  +650.656, Z    +0.000, E1   -14.835, E3 +149112.622}
SPL {X  -160.000, Y  +653.134, Z    +0.000, E1   -14.827, E3 +149132.549}
SPL {X  -160.000, Y  +655.670, Z    +0.000, E1   -14.841, E3 +149152.843}
SPL {X  -160.000, Y  +658.349, Z    +0.000, E1   -14.842, E3 +149174.318}
SPL {X  -160.000, Y  +660.936, Z    +0.000, E1   -14.838, E3 +149195.070}
SPL {X  -160.000, Y  +663.567, Z    +0.000, E1   -14.845, E3 +149216.201}
SPL {X  -160.000, Y  +666.216, Z    +0.000, E1   -14.832, E3 +149237.517}
SPL {X  -159.997, Y  +668.731, Z    +0.000, E1   -14.834, E3 +149257.709}
SPL {X  -159.962, Y  +671.176, Z    +0.000, E1   -14.822, E3 +149277.420}
SPL {X  -159.895, Y  +673.507, Z    +0.000, E1   -14.821, E3 +149296.152}
SPL {X  -159.785, Y  +675.985, Z    +0.000, E1   -14.818, E3 +149316.153}
SPL {X  -159.627, Y  +678.622, Z    +0.000, E1   -14.804, E3 +149337.506}
SPL {X  -159.438, Y  +681.094, Z    +0.000, E1   -14.770, E3 +149357.677}
SPL {X  -159.262, Y  +683.054, Z    +0.000, E1   -14.719, E3 +149373.906}
ENDSPLINE

SPLINE
SPL {X  -159.661, Y  +678.114, Z    +0.000, E1    -9.575, E3 +149403.498}
SPL {X  -159.942, Y  +672.020, Z    +0.000, E1    -4.692, E3 +149422.125}
SPL {X  -160.000, Y  +664.971, Z    +0.000, E1    +0.516, E3 +149441.675}
SPL {X  -160.000, Y  +660.032, Z    +0.000, E1    +3.995, E3 +149453.618}
SPL {X  -160.000, Y  +652.280, Z    +0.000, E1    +8.913, E3 +149472.133}
SPL {X  -160.000, Y  +644.147, Z    +0.000, E1   +13.158, E3 +149495.683}
SPL {X  -160.000, Y  +641.594, Z    +0.000, E1   +13.488, E3 +149514.124}
SPL {X  -160.000, Y  +639.799, Z    +0.000, E1   +13.486, E3 +149530.034}
SPL {X  -160.000, Y  +637.896, Z    +0.000, E1   +13.493, E3 +149546.849}
SPL {X  -160.000, Y  +635.832, Z    +0.000, E1   +13.499, E3 +149565.108}
SPL {X  -160.000, Y  +633.839, Z    +0.000, E1   +13.489, E3 +149582.797}
SPL {X  -160.000, Y  +631.625, Z    +0.000, E1   +13.508, E3 +149602.338}
SPL {X  -160.000, Y  +629.417, Z    +0.000, E1   +13.491, E3 +149621.949}
SPL {X  -160.000, Y  +627.180, Z    +0.000, E1   +13.508, E3 +149641.703}
SPL {X  -160.000, Y  +624.970, Z    +0.000, E1   +13.490, E3 +149661.353}
SPL {X  -160.000, Y  +623.020, Z    +0.000, E1   +13.491, E3 +149678.583}
SPL {X  -160.000, Y  +620.888, Z    +0.000, E1   +13.501, E3 +149697.445}
SPL {X  -160.000, Y  +618.790, Z    +0.000, E1   +13.488, E3 +149716.068}
SPL {X  -160.000, Y  +616.631, Z    +0.000, E1   +13.504, E3 +149735.121}
SPL {X  -160.000, Y  +614.230, Z    +0.000, E1   +13.510, E3 +149756.317}
SPL {X  -160.000, Y  +612.132, Z    +0.000, E1   +13.485, E3 +149775.033}
SPL {X  -160.000, Y  +610.405, Z    +0.000, E1   +13.477, E3 +149790.407}
SPL {X  -160.000, Y  +608.437, Z    +0.000, E1   +13.502, E3 +149807.662}
SPL {X  -160.000, Y  +606.281, Z    +0.000, E1   +13.502, E3 +149826.680}
SPL {X  -160.000, Y  +604.124, Z    +0.000, E1   +13.513, E3 +149845.735}
SPL {X  -160.000, Y  +601.878, Z    +0.000, E1   +13.505, E3 +149865.632}
SPL {X  -160.000, Y  +599.648, Z    +0.000, E1   +13.506, E3 +149885.409}
SPL {X  -160.000, Y  +597.673, Z    +0.000, E1   +13.479, E3 +149903.083}
SPL {X  -160.000, Y  +595.601, Z    +0.000, E1   +13.499, E3 +149921.366}
SPL {X  -160.000, Y  +593.187, Z    +0.000, E1   +13.500, E3 +149942.746}
SPL {X  -160.000, Y  +591.079, Z    +0.000, E1   +13.483, E3 +149961.472}
SPL {X  -160.000, Y  +589.151, Z    +0.000, E1   +13.489, E3 +149978.523}
SPL {X  -160.000, Y  +586.908, Z    +0.000, E1   +13.501, E3 +149998.368}
SPL {X  -160.000, Y  +584.660, Z    +0.000, E1   +13.490, E3 +150018.310}
SPL {X  -160.000, Y  +582.409, Z    +0.000, E1   +13.499, E3 +150038.228}
SPL {X  -160.000, Y  +580.150, Z    +0.000, E1   +13.490, E3 +150058.275}
SPL {X  -160.000, Y  +577.953, Z    +0.000, E1   +13.493, E3 +150077.733}
SPL {X  -160.000, Y  +575.630, Z    +0.000, E1   +13.502, E3 +150098.217}
SPL {X  -160.000, Y  +573.418, Z    +0.000, E1   +13.502, E3 +150117.725}
SPL {X  -160.000, Y  +571.226, Z    +0.000, E1   +13.520, E3 +150136.934}
SPL {X  -160.000, Y  +569.166, Z    +0.000, E1   +13.512, E3 +150155.124}
SPL {X  -160.000, Y  +567.275, Z    +0.000, E1   +13.517, E3 +150171.791}
SPL {X  -160.000, Y  +565.259, Z    +0.000, E1   +13.523, E3 +150189.581}
SPL {X  -160.000, Y  +563.305, Z    +0.000, E1   +13.512, E3 +150206.919}
SPL {X  -160.000, Y  +561.240, Z    +0.000, E1   +13.521, E3 +150225.180}
SPL {X  -160.000, Y  +558.881, Z    +0.000, E1   +13.524, E3 +150246.023}
SPL {X  -160.000, Y  +556.697, Z    +0.000, E1   +13.510, E3 +150265.409}
SPL {X  -160.000, Y  +554.624, Z    +0.000, E1   +13.512, E3 +150283.740}
SPL {X  -160.000, Y  +552.465, Z    +0.000, E1   +13.514, E3 +150302.824}
SPL {X  -160.000, Y  +550.315, Z    +0.000, E1   +13.514, E3 +150321.818}
SPL {X  -160.000, Y  +548.056, Z    +0.000, E1   +13.519, E3 +150341.819}
SPL {X  -160.000, Y  +545.826, Z    +0.000, E1   +13.501, E3 +150361.696}
SPL {X  -160.000, Y  +543.677, Z    +0.000, E1   +13.502, E3 +150380.754}
SPL {X  -160.000, Y  +541.664, Z    +0.000, E1   +13.489, E3 +150398.640}
SPL {X  -160.000, Y  +539.659, Z    +0.000, E1   +13.494, E3 +150416.400}
SPL {X  -160.000, Y  +537.370, Z    +0.000, E1   +13.501, E3 +150436.639}
SPL {X  -160.000, Y  +535.056, Z    +0.000, E1   +13.506, E3 +150457.034}
SPL {X  -160.000, Y  +532.975, Z    +0.000, E1   +13.494, E3 +150475.521}
SPL {X  -160.000, Y  +530.925, Z    +0.000, E1   +13.499, E3 +150493.683}
SPL {X  -160.000, Y  +528.768, Z    +0.000, E1   +13.498, E3 +150512.784}
SPL {X  -160.000, Y  +526.547, Z    +0.000, E1   +13.499, E3 +150532.453}
SPL {X  -160.000, Y  +523.964, Z    +0.000, E1   +13.742, E3 +150551.957}
SPL {X  -160.000, Y  +513.971, Z    +0.000, E1   +18.644, E3 +150570.869}
SPL {X  -160.000, Y  +513.562, Z    +0.000, E1   +16.972, E3 +150590.746}
SPL {X  -160.000, Y  +513.358, Z    +0.000, E1   +15.267, E3 +150611.018}
SPL {X  -160.000, Y  +512.244, Z    +0.000, E1   +14.473, E3 +150629.474}
SPL {X  -160.000, Y  +509.675, Z    +0.000, E1   +14.481, E3 +150650.618}
SPL {X  -160.000, Y  +507.162, Z    +0.000, E1   +14.470, E3 +150671.358}
SPL {X  -160.000, Y  +504.735, Z    +0.000, E1   +14.473, E3 +150691.329}
SPL {X  -160.000, Y  +502.261, Z    +0.000, E1   +14.476, E3 +150711.665}
SPL {X  -160.000, Y  +499.798, Z    +0.000, E1   +14.482, E3 +150731.868}
SPL {X  -160.000, Y  +497.435, Z    +0.000, E1   +14.476, E3 +150751.344}
SPL {X  -160.000, Y  +495.089, Z    +0.000, E1   +14.475, E3 +150770.711}
SPL {X  -160.000, Y  +492.764, Z    +0.000, E1   +14.469, E3 +150789.883}
SPL {X  -160.000, Y  +490.292, Z    +0.000, E1   +14.476, E3 +150810.283}
SPL {X  -160.000, Y  +487.641, Z    +0.000, E1   +14.470, E3 +150832.180}
SPL {X  -160.000, Y  +485.054, Z    +0.000, E1   +14.460, E3 +150853.622}
SPL {X  -160.000, Y  +482.421, Z    +0.000, E1   +14.461, E3 +150875.341}
SPL {X  -160.000, Y  +480.000, Z    +0.000, E1   +14.451, E3 +150895.305}
SPL {X  -160.000, Y  +477.551, Z    +0.000, E1   +14.466, E3 +150915.433}
SPL {X  -160.000, Y  +475.253, Z    +0.000, E1   +14.450, E3 +150934.407}
SPL {X  -160.000, Y  +473.070, Z    +0.000, E1   +14.454, E3 +150952.428}
SPL {X  -160.000, Y  +470.603, Z    +0.000, E1   +14.464, E3 +150972.728}
SPL {X  -160.000, Y  +468.243, Z    +0.000, E1   +14.458, E3 +150992.128}
SPL {X  -160.000, Y  +465.791, Z    +0.000, E1   +14.475, E3 +151012.272}
SPL {X  -160.000, Y  +463.103, Z    +0.000, E1   +14.474, E3 +151034.421}
SPL {X  -160.000, Y  +460.743, Z    +0.000, E1   +14.465, E3 +151053.829}
SPL {X  -160.000, Y  +458.292, Z    +0.000, E1   +14.492, E3 +151073.828}
SPL {X  -160.000, Y  +455.874, Z    +0.000, E1   +14.484, E3 +151093.686}
SPL {X  -160.000, Y  +453.555, Z    +0.000, E1   +14.488, E3 +151112.765}
SPL {X  -160.000, Y  +451.093, Z    +0.000, E1   +14.485, E3 +151133.077}
SPL {X  -160.000, Y  +448.700, Z    +0.000, E1   +14.483, E3 +151152.767}
SPL {X  -160.000, Y  +446.277, Z    +0.000, E1   +14.485, E3 +151172.690}
SPL {X  -160.000, Y  +443.879, Z    +0.000, E1   +14.485, E3 +151192.428}
SPL {X  -160.000, Y  +441.447, Z    +0.000, E1   +14.485, E3 +151212.436}
SPL {X  -160.000, Y  +439.006, Z    +0.000, E1   +14.488, E3 +151232.519}
SPL {X  -160.000, Y  +436.311, Z    +0.000, E1   +14.498, E3 +151254.678}
SPL {X  -160.000, Y  +433.559, Z    +0.000, E1   +14.491, E3 +151277.347}
SPL {X  -160.000, Y  +431.162, Z    +0.000, E1   +14.479, E3 +151297.098}
SPL {X  -160.000, Y  +429.152, Z    +0.000, E1   +14.469, E3 +151313.680}
SPL {X  -160.000, Y  +426.863, Z    +0.000, E1   +14.490, E3 +151332.459}
SPL {X  -160.000, Y  +424.653, Z    +0.000, E1   +14.467, E3 +151350.718}
SPL {X  -160.000, Y  +422.337, Z    +0.000, E1   +14.492, E3 +151369.702}
SPL {X  -160.000, Y  +419.639, Z    +0.000, E1   +14.504, E3 +151391.742}
SPL {X  -160.000, Y  +417.127, Z    +0.000, E1   +14.501, E3 +151412.333}
SPL {X  -160.000, Y  +414.849, Z    +0.000, E1   +14.496, E3 +151431.067}
SPL {X  -160.000, Y  +412.396, Z    +0.000, E1   +14.505, E3 +151451.256}
SPL {X  -160.000, Y  +409.815, Z    +0.000, E1   +14.498, E3 +151472.511}
SPL {X  -160.000, Y  +407.614, Z    +0.000, E1   +14.484, E3 +151490.636}
SPL {X  -160.000, Y  +405.406, Z    +0.000, E1   +14.501, E3 +151508.699}
SPL {X  -160.000, Y  +402.958, Z    +0.000, E1   +14.500, E3 +151528.869}
SPL {X  -160.000, Y  +400.690, Z    +0.000, E1   +14.484, E3 +151547.581}
SPL {X  -160.000, Y  +398.391, Z    +0.000, E1   +14.502, E3 +151566.407}
SPL {X  -160.000, Y  +395.999, Z    +0.000, E1   +14.484, E3 +151586.196}
SPL {X  -160.000, Y  +393.685, Z    +0.000, E1   +14.486, E3 +151605.269}
SPL {X  -159.999, Y  +391.313, Z    +0.000, E1   +14.479, E3 +151624.851}
SPL {X  -159.970, Y  +388.900, Z    +0.000, E1   +14.480, E3 +151644.735}
SPL {X  -159.903, Y  +386.417, Z    +0.000, E1   +14.475, E3 +151665.240}
SPL {X  -159.796, Y  +383.921, Z    +0.000, E1   +14.466, E3 +151685.896}
SPL {X  -159.651, Y  +381.443, Z    +0.000, E1   +14.453, E3 +151706.443}
SPL {X  -159.474, Y  +379.042, Z    +0.000, E1   +14.434, E3 +151726.407}
SPL {X  -159.316, Y  +377.219, Z    +0.000, E1   +14.400, E3 +151741.636}
ENDSPLINE

SPLINE
SPL {X  -159.452, Y  +378.767, Z    +0.000, E1   +11.887, E3 +151762.625}
SPL {X  -159.840, Y  +384.856, Z    +0.000, E1    +7.126, E3 +151781.597}
SPL {X  -159.991, Y  +390.336, Z    +0.000, E1    +2.803, E3 +151795.419}
SPL {X  -160.000, Y  +403.532, Z    +0.000, E1    -6.523, E3 +151813.140}
SPL {X  -160.000, Y  +409.023, Z    +0.000, E1   -10.003, E3 +151823.914}
SPL {X  -160.000, Y  +418.032, Z    +0.000, E1   -14.569, E3 +151848.773}
SPL {X  -160.000, Y  +420.561, Z    +0.000, E1   -14.816, E3 +151866.253}
SPL {X  -160.000, Y  +422.801, Z    +0.000, E1   -14.823, E3 +151884.201}
SPL {X  -160.000, Y  +425.518, Z    +0.000, E1   -14.845, E3 +151905.976}
SPL {X  -160.000, Y  +428.688, Z    +0.000, E1   -14.854, E3 +151931.384}
SPL {X  -160.000, Y  +431.971, Z    +0.000, E1   -14.849, E3 +151957.853}
SPL {X  -160.000, Y  +435.345, Z    +0.000, E1   -14.857, E3 +151984.903}
SPL {X  -160.000, Y  +438.732, Z    +0.000, E1   -14.858, E3 +152012.051}
SPL {X  -160.000, Y  +441.925, Z    +0.000, E1   -14.848, E3 +152037.722}
SPL {X  -160.000, Y  +444.299, Z    +0.000, E1   -14.809, E3 +152056.906}
SPL {X  -160.000, Y  +446.229, Z    +0.000, E1   -14.820, E3 +152072.325}
SPL {X  -160.000, Y  +448.987, Z    +0.000, E1   -14.868, E3 +152094.262}
SPL {X  -160.000, Y  +452.351, Z    +0.000, E1   -14.871, E3 +152121.238}
SPL {X  -160.000, Y  +455.709, Z    +0.000, E1   -14.880, E3 +152148.052}
SPL {X  -160.000, Y  +458.189, Z    +0.000, E1   -14.832, E3 +152168.054}
SPL {X  -160.000, Y  +459.885, Z    +0.000, E1   -14.825, E3 +152181.725}
SPL {X  -160.000, Y  +462.438, Z    +0.000, E1   -14.868, E3 +152202.135}
SPL {X  -160.000, Y  +465.575, Z    +0.000, E1   -14.849, E3 +152227.443}
SPL {X  -160.000, Y  +468.581, Z    +0.000, E1   -14.841, E3 +152251.675}
SPL {X  -160.000, Y  +471.795, Z    +0.000, E1   -14.854, E3 +152277.463}
SPL {X  -160.000, Y  +475.138, Z    +0.000, E1   -14.853, E3 +152304.313}
SPL {X  -160.000, Y  +477.981, Z    +0.000, E1   -14.823, E3 +152327.233}
SPL {X  -160.000, Y  +480.658, Z    +0.000, E1   -14.835, E3 +152348.709}
SPL {X  -160.000, Y  +483.534, Z    +0.000, E1   -14.838, E3 +152371.804}
SPL {X  -160.000, Y  +486.226, Z    +0.000, E1   -14.823, E3 +152393.469}
SPL {X  -160.000, Y  +488.751, Z    +0.000, E1   -14.827, E3 +152413.742}
SPL {X  -160.000, Y  +491.612, Z    +0.000, E1   -14.844, E3 +152436.664}
SPL {X  -160.000, Y  +494.417, Z    +0.000, E1   -14.827, E3 +152459.255}
SPL {X  -160.000, Y  +496.961, Z    +0.000, E1   -14.824, E3 +152479.699}
SPL {X  -160.000, Y  +499.610, Z    +0.000, E1   -14.830, E3 +152500.972}
SPL {X  -160.000, Y  +502.268, Z    +0.000, E1   -14.832, E3 +152522.241}
SPL {X  -160.000, Y  +505.041, Z    +0.000, E1   -14.849, E3 +152544.403}
SPL {X  -160.000, Y  +507.743, Z    +0.000, E1   -14.842, E3 +152566.027}
SPL {X  -160.000, Y  +510.437, Z    +0.000, E1   -14.860, E3 +152587.541}
SPL {X  -160.000, Y  +513.179, Z    +0.000, E1   -14.849, E3 +152609.588}
SPL {X  -160.000, Y  +515.613, Z    +0.000, E1   -14.829, E3 +152629.259}
SPL {X  -160.000, Y  +518.188, Z    +0.000, E1   -14.845, E3 +152649.888}
SPL {X  -160.000, Y  +520.790, Z    +0.000, E1   -14.839, E3 +152670.717}
SPL {X  -160.000, Y  +523.469, Z    +0.000, E1   -14.855, E3 +152692.165}
SPL {X  -160.000, Y  +526.403, Z    +0.000, E1   -14.858, E3 +152715.702}
SPL {X  -160.000, Y  +529.266, Z    +0.000, E1   -14.848, E3 +152738.709}
SPL {X  -160.000, Y  +531.688, Z    +0.000, E1   -14.826, E3 +152758.259}
SPL {X  -160.000, Y  +534.214, Z    +0.000, E1   -14.841, E3 +152778.522}
SPL {X  -160.000, Y  +537.002, Z    +0.000, E1   -14.839, E3 +152800.940}
SPL {X  -160.000, Y  +539.729, Z    +0.000, E1   -14.840, E3 +152822.751}
SPL {X  -160.000, Y  +542.408, Z    +0.000, E1   -14.839, E3 +152844.304}
SPL {X  -160.000, Y  +545.014, Z    +0.000, E1   -14.831, E3 +152865.250}
SPL {X  -160.000, Y  +547.659, Z    +0.000, E1   -14.839, E3 +152886.464}
SPL {X  -160.000, Y  +550.215, Z    +0.000, E1   -14.827, E3 +152907.029}
SPL {X  -160.000, Y  +552.762, Z    +0.000, E1   -14.836, E3 +152927.447}
SPL {X  -160.000, Y  +555.331, Z    +0.000, E1   -14.837, E3 +152947.988}
SPL {X  -160.000, Y  +558.235, Z    +0.000, E1   -14.869, E3 +152971.152}
SPL {X  -160.000, Y  +561.088, Z    +0.000, E1   -14.848, E3 +152994.070}
SPL {X  -160.000, Y  +563.693, Z    +0.000, E1   -14.852, E3 +153014.931}
SPL {X  -160.000, Y  +566.560, Z    +0.000, E1   -14.865, E3 +153037.909}
SPL {X  -160.000, Y  +569.305, Z    +0.000, E1   -14.848, E3 +153059.937}
SPL {X  -160.000, Y  +571.769, Z    +0.000, E1   -14.852, E3 +153079.683}
SPL {X  -160.000, Y  +574.366, Z    +0.000, E1   -14.855, E3 +153100.470}
SPL {X  -160.000, Y  +577.037, Z    +0.000, E1   -14.859, E3 +153121.869}
SPL {X  -160.000, Y  +579.855, Z    +0.000, E1   -14.869, E3 +153144.397}
SPL {X  -160.000, Y  +582.456, Z    +0.000, E1   -14.854, E3 +153165.257}
SPL {X  -160.000, Y  +585.083, Z    +0.000, E1   -14.866, E3 +153186.306}
SPL {X  -160.000, Y  +587.675, Z    +0.000, E1   -14.853, E3 +153207.097}
SPL {X  -160.000, Y  +590.216, Z    +0.000, E1   -14.864, E3 +153227.416}
SPL {X  -160.000, Y  +592.848, Z    +0.000, E1   -14.865, E3 +153248.467}
SPL {X  -160.000, Y  +595.342, Z    +0.000, E1   -14.848, E3 +153268.645}
SPL {X  -160.000, Y  +597.995, Z    +0.000, E1   -14.848, E3 +153289.985}
SPL {X  -160.000, Y  +600.731, Z    +0.000, E1   -14.846, E3 +153311.936}
SPL {X  -160.000, Y  +603.404, Z    +0.000, E1   -14.846, E3 +153333.372}
SPL {X  -160.000, Y  +605.923, Z    +0.000, E1   -14.838, E3 +153353.613}
SPL {X  -160.000, Y  +608.492, Z    +0.000, E1   -14.846, E3 +153374.217}
SPL {X  -160.000, Y  +611.345, Z    +0.000, E1   -14.856, E3 +153397.075}
SPL {X  -160.000, Y  +614.087, Z    +0.000, E1   -14.839, E3 +153419.134}
SPL {X  -160.000, Y  +616.566, Z    +0.000, E1   -14.839, E3 +153439.028}
SPL {X  -160.000, Y  +619.350, Z    +0.000, E1   -14.855, E3 +153461.316}
SPL {X  -160.000, Y  +622.198, Z    +0.000, E1   -14.846, E3 +153484.201}
SPL {X  -160.000, Y  +624.642, Z    +0.000, E1   -14.829, E3 +153503.873}
SPL {X  -160.000, Y  +627.119, Z    +0.000, E1   -14.843, E3 +153523.713}
SPL {X  -160.000, Y  +629.682, Z    +0.000, E1   -14.838, E3 +153544.282}
SPL {X  -160.000, Y  +632.223, Z    +0.000, E1   -14.841, E3 +153564.673}
SPL {X  -160.000, Y  +634.941, Z    +0.000, E1   -14.846, E3 +153586.471}
SPL {X  -160.000, Y  +637.723, Z    +0.000, E1   -14.844, E3 +153608.815}
SPL {X  -160.000, Y  +640.315, Z    +0.000, E1   -14.836, E3 +153629.613}
SPL {X  -160.000, Y  +643.085, Z    +0.000, E1   -14.865, E3 +153651.664}
SPL {X  -160.000, Y  +645.845, Z    +0.000, E1   -14.848, E3 +153673.852}
SPL {X  -160.000, Y  +648.229, Z    +0.000, E1   -14.834, E3 +153693.062}
SPL {X  -160.000, Y  +650.656, Z    +0.000, E1   -14.835, E3 +153712.619}
SPL {X  -160.000, Y  +653.134, Z    +0.000, E1   -14.827, E3 +153732.545}
SPL {X  -160.000, Y  +655.670, Z    +0.000, E1   -14.841, E3 +153752.840}
SPL {X  -160.000, Y  +658.349, Z    +0.000, E1   -14.842, E3 +153774.315}
SPL {X  -160.000, Y  +660.936, Z    +0.000, E1   -14.838, E3 +153795.067}
SPL {X  -160.000, Y  +663.567, Z    +0.000, E1   -14.845, E3 +153816.198}
SPL {X  -160.000, Y  +666.216, Z    +0.000, E1   -14.832, E3 +153837.514}
SPL {X  -159.997, Y  +668.731, Z    +0.000, E1   -14.834, E3 +153857.706}
SPL {X  -159.962, Y  +671.176, Z    +0.000, E1   -14.822, E3 +153877.417}
SPL {X  -159.895, Y  +673.507, Z    +0.000, E1   -14.821, E3 +153896.148}
SPL {X  -159.785, Y  +675.985, Z    +0.000, E1   -14.818, E3 +153916.150}
SPL {X  -159.627, Y  +678.622, Z    +0.000, E1   -14.804, E3 +153937.503}
SPL {X  -159.438, Y  +681.094, Z    +0.000, E1   -14.770, E3 +153957.674}
SPL {X  -159.262, Y  +683.054, Z    +0.000, E1   -14.719, E3 +153973.903}
ENDSPLINE

SPLINE
SPL {X  -159.661, Y  +678.114, Z    +0.000, E1    -9.575, E3 +154003.495}
SPL {X  -159.942, Y  +672.020, Z    +0.000, E1    -4.692, E3 +154022.121}
SPL {X  -160.000, Y  +664.971, Z    +0.000, E1    +0.516, E3 +154041.672}
SPL {X  -160.000, Y  +660.032, Z    +0.000, E1    +3.995, E3 +154053.615}
SPL {X  -160.000, Y  +652.280, Z    +0.000, E1    +8.913, E3 +154072.130}
SPL {X  -160.000, Y  +644.147, Z    +0.000, E1   +13.158, E3 +154095.680}
SPL {X  -160.000, Y  +641.594, Z    +0.000, E1   +13.488, E3 +154114.121}
SPL {X  -160.000, Y  +639.799, Z    +0.000, E1   +13.486, E3 +154130.031}
SPL {X  -160.000, Y  +637.896, Z    +0.000, E1   +13.493, E3 +154146.846}
SPL {X  -160.000, Y  +635.832, Z    +0.000, E1   +13.499, E3 +154165.105}
SPL {X  -160.000, Y  +633.839, Z    +0.000, E1   +13.489, E3 +154182.794}
SPL {X  -160.000, Y  +631.625, Z    +0.000, E1   +13.508, E3 +154202.334}
SPL {X  -160.000, Y  +629.417, Z    +0.000, E1   +13.491, E3 +154221.946}
SPL {X  -160.000, Y  +627.180, Z    +0.000, E1   +13.508, E3 +154241.700}
SPL {X  -160.000, Y  +624.970, Z    +0.000, E1   +13.490, E3 +154261.350}
SPL {X  -160.000, Y  +623.020, Z    +0.000, E1   +13.491, E3 +154278.580}
SPL {X  -160.000, Y  +620.888, Z    +0.000, E1   +13.501, E3 +154297.442}
SPL {X  -160.000, Y  +618.790, Z    +0.000, E1   +13.488, E3 +154316.064}
SPL {X  -160.000, Y  +616.631, Z    +0.000, E1   +13.504, E3 +154335.118}
SPL {X  -160.000, Y  +614.230, Z    +0.000, E1   +13.510, E3 +154356.314}
SPL {X  -160.000, Y  +612.132, Z    +0.000, E1   +13.485, E3 +154375.030}
SPL {X  -160.000, Y  +610.405, Z    +0.000, E1   +13.477, E3 +154390.404}
SPL {X  -160.000, Y  +608.437, Z    +0.000, E1   +13.502, E3 +154407.659}
SPL {X  -160.000, Y  +606.281, Z    +0.000, E1   +13.502, E3 +154426.677}
SPL {X  -160.000, Y  +604.124, Z    +0.000, E1   +13.513, E3 +154445.732}
SPL {X  -160.000, Y  +601.878, Z    +0.000, E1   +13.505, E3 +154465.629}
SPL {X  -160.000, Y  +599.648, Z    +0.000, E1   +13.506, E3 +154485.406}
SPL {X  -160.000, Y  +597.673, Z    +0.000, E1   +13.479, E3 +154503.079}
SPL {X  -160.000, Y  +595.601, Z    +0.000, E1   +13.499, E3 +154521.363}
SPL {X  -160.000, Y  +593.187, Z    +0.000, E1   +13.500, E3 +154542.743}
SPL {X  -160.000, Y  +591.079, Z    +0.000, E1   +13.483, E3 +154561.469}
SPL {X  -160.000, Y  +589.151, Z    +0.000, E1   +13.489, E3 +154578.520}
SPL {X  -160.000, Y  +586.908, Z    +0.000, E1   +13.501, E3 +154598.365}
SPL {X  -160.000, Y  +584.660, Z    +0.000, E1   +13.490, E3 +154618.307}
SPL {X  -160.000, Y  +582.409, Z    +0.000, E1   +13.499, E3 +154638.225}
SPL {X  -160.000, Y  +580.150, Z    +0.000, E1   +13.490, E3 +154658.272}
SPL {X  -160.000, Y  +577.953, Z    +0.000, E1   +13.493, E3 +154677.730}
SPL {X  -160.000, Y  +575.630, Z    +0.000, E1   +13.502, E3 +154698.214}
SPL {X  -160.000, Y  +573.418, Z    +0.000, E1   +13.502, E3 +154717.722}
SPL {X  -160.000, Y  +571.226, Z    +0.000, E1   +13.520, E3 +154736.931}
SPL {X  -160.000, Y  +569.166, Z    +0.000, E1   +13.512, E3 +154755.121}
SPL {X  -160.000, Y  +567.275, Z    +0.000, E1   +13.517, E3 +154771.788}
SPL {X  -160.000, Y  +565.259, Z    +0.000, E1   +13.523, E3 +154789.577}
SPL {X  -160.000, Y  +563.305, Z    +0.000, E1   +13.512, E3 +154806.916}
SPL {X  -160.000, Y  +561.240, Z    +0.000, E1   +13.521, E3 +154825.177}
SPL {X  -160.000, Y  +558.881, Z    +0.000, E1   +13.524, E3 +154846.020}
SPL {X  -160.000, Y  +556.697, Z    +0.000, E1   +13.510, E3 +154865.406}
SPL {X  -160.000, Y  +554.624, Z    +0.000, E1   +13.512, E3 +154883.737}
SPL {X  -160.000, Y  +552.465, Z    +0.000, E1   +13.514, E3 +154902.821}
SPL {X  -160.000, Y  +550.315, Z    +0.000, E1   +13.514, E3 +154921.814}
SPL {X  -160.000, Y  +548.056, Z    +0.000, E1   +13.519, E3 +154941.815}
SPL {X  -160.000, Y  +545.826, Z    +0.000, E1   +13.501, E3 +154961.693}
SPL {X  -160.000, Y  +543.677, Z    +0.000, E1   +13.502, E3 +154980.751}
SPL {X  -160.000, Y  +541.664, Z    +0.000, E1   +13.489, E3 +154998.636}
SPL {X  -160.000, Y  +539.659, Z    +0.000, E1   +13.494, E3 +155016.397}
SPL {X  -160.000, Y  +537.370, Z    +0.000, E1   +13.501, E3 +155036.636}
SPL {X  -160.000, Y  +535.056, Z    +0.000, E1   +13.506, E3 +155057.031}
SPL {X  -160.000, Y  +532.975, Z    +0.000, E1   +13.494, E3 +155075.518}
SPL {X  -160.000, Y  +530.925, Z    +0.000, E1   +13.499, E3 +155093.680}
SPL {X  -160.000, Y  +528.768, Z    +0.000, E1   +13.498, E3 +155112.781}
SPL {X  -160.000, Y  +526.547, Z    +0.000, E1   +13.499, E3 +155132.450}
SPL {X  -160.000, Y  +523.964, Z    +0.000, E1   +13.742, E3 +155151.954}
SPL {X  -160.000, Y  +513.971, Z    +0.000, E1   +18.644, E3 +155170.866}
SPL {X  -160.000, Y  +513.562, Z    +0.000, E1   +16.972, E3 +155190.743}
SPL {X  -160.000, Y  +513.358, Z    +0.000, E1   +15.267, E3 +155211.015}
SPL {X  -160.000, Y  +512.244, Z    +0.000, E1   +14.473, E3 +155229.471}
SPL {X  -160.000, Y  +509.675, Z    +0.000, E1   +14.481, E3 +155250.615}
SPL {X  -160.000, Y  +507.162, Z    +0.000, E1   +14.470, E3 +155271.355}
SPL {X  -160.000, Y  +504.735, Z    +0.000, E1   +14.473, E3 +155291.326}
SPL {X  -160.000, Y  +502.261, Z    +0.000, E1   +14.476, E3 +155311.662}
SPL {X  -160.000, Y  +499.798, Z    +0.000, E1   +14.482, E3 +155331.864}
SPL {X  -160.000, Y  +497.435, Z    +0.000, E1   +14.476, E3 +155351.341}
SPL {X  -160.000, Y  +495.089, Z    +0.000, E1   +14.475, E3 +155370.708}
SPL {X  -160.000, Y  +492.764, Z    +0.000, E1   +14.469, E3 +155389.879}
SPL {X  -160.000, Y  +490.292, Z    +0.000, E1   +14.476, E3 +155410.280}
SPL {X  -160.000, Y  +487.641, Z    +0.000, E1   +14.470, E3 +155432.176}
SPL {X  -160.000, Y  +485.054, Z    +0.000, E1   +14.460, E3 +155453.619}
SPL {X  -160.000, Y  +482.421, Z    +0.000, E1   +14.461, E3 +155475.337}
SPL {X  -160.000, Y  +480.000, Z    +0.000, E1   +14.451, E3 +155495.302}
SPL {X  -160.000, Y  +477.551, Z    +0.000, E1   +14.466, E3 +155515.430}
SPL {X  -160.000, Y  +475.253, Z    +0.000, E1   +14.450, E3 +155534.404}
SPL {X  -160.000, Y  +473.070, Z    +0.000, E1   +14.454, E3 +155552.425}
SPL {X  -160.000, Y  +470.603, Z    +0.000, E1   +14.464, E3 +155572.725}
SPL {X  -160.000, Y  +468.243, Z    +0.000, E1   +14.458, E3 +155592.125}
SPL {X  -160.000, Y  +465.791, Z    +0.000, E1   +14.475, E3 +155612.269}
SPL {X  -160.000, Y  +463.103, Z    +0.000, E1   +14.474, E3 +155634.417}
SPL {X  -160.000, Y  +460.743, Z    +0.000, E1   +14.465, E3 +155653.826}
SPL {X  -160.000, Y  +458.292, Z    +0.000, E1   +14.492, E3 +155673.825}
SPL {X  -160.000, Y  +455.874, Z    +0.000, E1   +14.484, E3 +155693.683}
SPL {X  -160.000, Y  +453.555, Z    +0.000, E1   +14.488, E3 +155712.762}
SPL {X  -160.000, Y  +451.093, Z    +0.000, E1   +14.485, E3 +155733.074}
SPL {X  -160.000, Y  +448.700, Z    +0.000, E1   +14.483, E3 +155752.763}
SPL {X  -160.000, Y  +446.277, Z    +0.000, E1   +14.485, E3 +155772.687}
SPL {X  -160.000, Y  +443.879, Z    +0.000, E1   +14.485, E3 +155792.425}
SPL {X  -160.000, Y  +441.447, Z    +0.000, E1   +14.485, E3 +155812.432}
SPL {X  -160.000, Y  +439.006, Z    +0.000, E1   +14.488, E3 +155832.515}
SPL {X  -160.000, Y  +436.311, Z    +0.000, E1   +14.498, E3 +155854.674}
SPL {X  -160.000, Y  +433.559, Z    +0.000, E1   +14.491, E3 +155877.344}
SPL {X  -160.000, Y  +431.162, Z    +0.000, E1   +14.479, E3 +155897.095}
SPL {X  -160.000, Y  +429.152, Z    +0.000, E1   +14.469, E3 +155913.676}
SPL {X  -160.000, Y  +426.863, Z    +0.000, E1   +14.490, E3 +155932.455}
SPL {X  -160.000, Y  +424.653, Z    +0.000, E1   +14.467, E3 +155950.715}
SPL {X  -160.000, Y  +422.337, Z    +0.000, E1   +14.492, E3 +155969.699}
SPL {X  -160.000, Y  +419.639, Z    +0.000, E1   +14.504, E3 +155991.739}
SPL {X  -160.000, Y  +417.127, Z    +0.000, E1   +14.501, E3 +156012.330}
SPL {X  -160.000, Y  +414.849, Z    +0.000, E1   +14.496, E3 +156031.064}
SPL {X  -160.000, Y  +412.396, Z    +0.000, E1   +14.505, E3 +156051.253}
SPL {X  -160.000, Y  +409.815, Z    +0.000, E1   +14.498, E3 +156072.507}
SPL {X  -160.000, Y  +407.614, Z    +0.000, E1   +14.484, E3 +156090.633}
SPL {X  -160.000, Y  +405.406, Z    +0.000, E1   +14.501, E3 +156108.695}
SPL {X  -160.000, Y  +402.958, Z    +0.000, E1   +14.500, E3 +156128.866}
SPL {X  -160.000, Y  +400.690, Z    +0.000, E1   +14.484, E3 +156147.577}
SPL {X  -160.000, Y  +398.391, Z    +0.000, E1   +14.502, E3 +156166.403}
SPL {X  -160.000, Y  +395.999, Z    +0.000, E1   +14.484, E3 +156186.193}
SPL {X  -160.000, Y  +393.685, Z    +0.000, E1   +14.486, E3 +156205.266}
SPL {X  -159.999, Y  +391.313, Z    +0.000, E1   +14.479, E3 +156224.847}
SPL {X  -159.970, Y  +388.900, Z    +0.000, E1   +14.480, E3 +156244.732}
SPL {X  -159.903, Y  +386.417, Z    +0.000, E1   +14.475, E3 +156265.237}
SPL {X  -159.796, Y  +383.921, Z    +0.000, E1   +14.466, E3 +156285.893}
SPL {X  -159.651, Y  +381.443, Z    +0.000, E1   +14.453, E3 +156306.440}
SPL {X  -159.474, Y  +379.042, Z    +0.000, E1   +14.434, E3 +156326.404}
SPL {X  -159.316, Y  +377.219, Z    +0.000, E1   +14.400, E3 +156341.633}
ENDSPLINE

